CASE _eState
OF
  E_PROGRESS.PROGRESS_INIT:
    IF Execute 
    THEN
      memset(ADR(_stMsg),0,SIZEOF(_stMsg));
      _nErrorId                     := 0;
      _rValue                       := 0;
      _eState                       := E_PROGRESS.PROGRESS_BUSY;
    END_IF
END_CASE
CASE _eState
OF
  E_PROGRESS.PROGRESS_BUSY:
    IF (_AxisRef.NcToPlc.AxisId <> 0)
    THEN
      _stMsg.eType                  := E_MessageType.eMessageVerbose;
      _stMsg.eDevice                := e_Device.Axis + (_AxisRef.NcToPlc.AxisId);
      _stMsg.eSubdevice             := e_Subdevice.AxisStartUp;
      _stMsg.iErrorNumber           := 0;
      _stMsg.sText                  := concat('StartUp NcAxisId: ', TO_STRING(_AxisRef.NcToPlc.AxisId));

      IF (_MessageLevel = E_MessageType.eMessageVerbose)
      THEN
        f_MessageSet(_stMsg);
      END_IF

      _eState                       := E_PROGRESS.PROGRESS_STARTUP;
    END_IF
END_CASE
CASE _eState
OF
  E_PROGRESS.PROGRESS_STARTUP:
    _fbADSRead(
              NETID                 := '', 
              PORT                  := 501, 
              IDXGRP                := (16#5000 + _AxisRef.NcToPlc.AxisId), 
              IDXOFFS               := 16#00000003, // offset for encoder type
              LEN                   := SIZEOF(_nEncoderType), 
              DESTADDR              := ADR(_nEncoderType),
              TMOUT                 := T#200MS,
              READ                  := FALSE);

    // clear required ADS information
    _sAxisName      := _sName       := 'NO NAME';
    _sEncoderType   := _sEncoder    := 'NO TYPE';
    _nEncoderType   := _uiEncType   :=  0;

    _eState                         := E_PROGRESS.PROGRESS_PREPARE;
END_CASE
CASE _eState
OF
  E_PROGRESS.PROGRESS_PREPARE:
    _fbADSRead(
              NETID                 := '', 
              PORT                  := 501, 
              IDXGRP                := (16#5000 + _AxisRef.NcToPlc.AxisId), 
              IDXOFFS               := 16#00000003, // offset for encoder type
              LEN                   := SIZEOF(_nEncoderType), 
              DESTADDR              := ADR(_nEncoderType),
              TMOUT                 := T#200MS,
              READ                  := TRUE);

    IF (_fbADSRead.ERR)
    THEN
      _nErrorId                     := _fbAdsRead.ERRID;

      _stMsg.eType                  := E_MessageType.eMessageError;
      _stMsg.eDevice                := e_Device.Axis + (_AxisRef.NcToPlc.AxisId);
      _stMsg.eSubdevice             := e_Subdevice.AxisStartUp;
      _stMsg.iErrorNumber           := _nErrorId;
      _stMsg.sText                  := 'StartUp Ads Error Read Encoder Type';

      f_MessageSet(_stMsg);
      _eState                       := E_PROGRESS.PROGRESS_ERROR;

    ELSIF (_nEncoderType <> 0)
    THEN
      _uiEncType  := _eEncoderType  := _nEncoderType;
      _sEncoder   := _sEncoderType  := TO_STRING(_eEncoderType);

      _stMsg.eType                  := E_MessageType.eMessageInfo;
      _stMsg.eDevice                := e_Device.Axis + (_AxisRef.NcToPlc.AxisId);
      _stMsg.eSubdevice             := e_Subdevice.AxisStartUp;
      _stMsg.iErrorNumber           := 0;
      _stMsg.sText                  := concat('Encoder Type: ', _sEncoder);

      IF (_MessageLevel > E_MessageType.eMessageError)
      THEN
        f_MessageSet(_stMsg);
      END_IF

      _eState                       := E_PROGRESS.PROGRESS_CHECK;
    END_IF
END_CASE
CASE _eState
OF
  E_PROGRESS.PROGRESS_CHECK:
    _fbADSRead(
            NETID                   := '', 
            PORT                    := 501, 
            IDXGRP                  := (16#4000 + _AxisRef.NcToPlc.AxisId), 
            IDXOFFS                 := 16#00000002, // offset for axis name
            LEN                     := SIZEOF(_sAxisName), 
            DESTADDR                := ADR(_sAxisName),
            READ                    := FALSE);

    _eState                         := E_PROGRESS.PROGRESS_OCCUPIED;
END_CASE
CASE _eState
OF
  E_PROGRESS.PROGRESS_OCCUPIED:
    _fbADSRead(
            NETID                   := '', 
            PORT                    := 501, 
            IDXGRP                  := (16#4000 + _AxisRef.NcToPlc.AxisId), 
            IDXOFFS                 := 16#00000002, // offset for axis name
            LEN                     := SIZEOF(_sAxisName), 
            DESTADDR                := ADR(_sAxisName),
            READ                    := TRUE);

    IF (_fbADSRead.ERR)
    THEN
      _nErrorId                     := _fbAdsRead.ERRID;

      _stMsg.eType                  := E_MessageType.eMessageError;
      _stMsg.eDevice                := e_Device.Axis + (_AxisRef.NcToPlc.AxisId);;
      _stMsg.eSubdevice             := e_Subdevice.AxisStartUp;
      _stMsg.iErrorNumber           := _nErrorId;
      _stMsg.sText                  := 'StartUp Ads Error Read Axis Name';

      f_MessageSet(_stMsg);
      _eState                       := E_PROGRESS.PROGRESS_ERROR;

    ELSIF (_sAxisName <> 'NO NAME')
    THEN
      _sName                        := _sAxisName;

      _stMsg.eType                  := E_MessageType.eMessageInfo;
      _stMsg.eDevice                := e_Device.Axis + (_AxisRef.NcToPlc.AxisId);;
      _stMsg.eSubdevice             := e_Subdevice.AxisStartUp;
      _stMsg.iErrorNumber           := 0;
      _stMsg.sText                  := concat('Axis Name: ', _sName);

      IF (_MessageLevel > E_MessageType.eMessageError)
      THEN
        f_MessageSet(_stMsg);
      END_IF

      _eState                       := E_PROGRESS.PROGRESS_WORKING;
    END_IF
END_CASE
CASE _eState
OF
  E_PROGRESS.PROGRESS_WORKING:
    _eState                         := E_PROGRESS.PROGRESS_DONE;
END_CASE

StartUp                             := _eState;
END_METHOD

METHOD Stop : E_PROGRESS
VAR_INPUT
  Execute           : BOOL;
  Dec               : LREAL;
  Jerk              : LREAL;

END_VAR
VAR_INST
  _eState           : E_PROGRESS;
  _rValue           : LREAL;
  _stMsg            : ST_Message;
END_VAR
IF NOT (__ISVALIDREF(_AxisRef)) THEN  Stop  := E_PROGRESS.PROGRESS_ERROR; RETURN; END_IF
IF NOT Execute THEN _eState := E_PROGRESS.PROGRESS_INIT; END_IF

CASE _eState
OF
  E_PROGRESS.PROGRESS_INIT:
    IF Execute 
    THEN
      memset(ADR(_stMsg),0,SIZEOF(_stMsg));
      _nErrorId                     := 0;
      _rValue                       := 0;
      _eState                       := E_PROGRESS.PROGRESS_BUSY;
    END_IF
END_CASE
CASE _eState
OF
  E_PROGRESS.PROGRESS_BUSY:
    _eState                         := E_PROGRESS.PROGRESS_OCCUPIED;
    _fbStop(
              Axis                  := _AxisRef, 
              Execute               := FALSE, 
              Deceleration          := Dec, 
              Jerk                  := Jerk);
END_CASE
CASE _eState
OF
  E_PROGRESS.PROGRESS_OCCUPIED:
    _fbStop(
              Axis                  := _AxisRef, 
              Execute               := TRUE, 
              Deceleration          := Dec, 
              Jerk                  := Jerk);

    IF _fbStop.Error
    THEN
        _nErrorId                   := _fbStop.ErrorID;

        _stMsg.eType                := E_MessageType.eMessageError;
        _stMsg.eDevice              := e_Device.Axis + (_AxisRef.NcToPlc.AxisId);
        _stMsg.eSubdevice           := e_SubDevice.fbStop;
        _stMsg.iErrorNumber         := _nErrorId;

        f_MessageSet(_stMsg);
        _fbStop(
              Axis                  := _AxisRef, 
              Execute               := FALSE);

      _eState                       := E_PROGRESS.PROGRESS_ERROR;

    ELSE
      IF _fbStop.Done OR
         _AxisRef.Status.NotMoving
      THEN
        _eState                     := E_PROGRESS.PROGRESS_WORKING;

      ELSIF _fbStop.CommandAborted
      THEN
        _eState                     := E_PROGRESS.PROGRESS_BUSY;
      END_IF
    END_IF
END_CASE
CASE _eState
OF
  E_PROGRESS.PROGRESS_WORKING:
    _fbStop(
              Axis                  := _AxisRef, 
              Execute               := FALSE);

    _eState                         := E_PROGRESS.PROGRESS_DONE;
END_CASE


Stop                                := _eState;
END_METHOD

METHOD Template : E_PROGRESS
VAR_INPUT
  Execute           : BOOL;
END_VAR
VAR_INST
  _eState           : E_PROGRESS;
  _rValue           : LREAL;
  _udiErr           : UDINT;
  _stMsg            : ST_Message;


END_VAR
IF NOT (__ISVALIDREF(_AxisRef)) THEN _eState := E_PROGRESS.ERROR; END_IF
IF NOT Execute THEN _eState := E_PROGRESS.INIT; END_IF

CASE _eState
OF
  E_PROGRESS.INIT:
    IF Execute 
    THEN
      memset(ADR(_stMsg),0,SIZEOF(_stMsg));
      _udiErr                       := 0;
      _rValue                       := 0;
      _eState                       := E_PROGRESS.BUSY;
    END_IF
END_CASE
CASE _eState
OF
  E_PROGRESS.BUSY:
    _eState                         := E_PROGRESS.STARTUP;
END_CASE
CASE _eState
OF
  E_PROGRESS.STARTUP:
    _eState                       := E_PROGRESS.PREPARE;
END_CASE
CASE _eState
OF
  E_PROGRESS.PREPARE:
    _eState                         := E_PROGRESS.READY;
END_CASE
CASE _eState
OF
  E_PROGRESS.READY:
    _eState                         := E_PROGRESS.WAITING;
END_CASE
CASE _eState
OF
  E_PROGRESS.WAITING:
    _eState                         := E_PROGRESS.WORKING;
END_CASE
CASE _eState
OF
  E_PROGRESS.WORKING:
    _eState                         := E_PROGRESS.DONE;
END_CASE

Template_1 := _eState;
END_METHOD

METHOD WriteParameter : E_PROGRESS
VAR_INPUT
  Execute           : BOOL;
  Value             : LREAL;
  ParameterNumber   : Tc2_MC2.MC_AxisParameter;
END_VAR
VAR_INST
  _eState           : E_PROGRESS;
  _nParameter       : Tc2_MC2.MC_AxisParameter;
  _rValue           : LREAL;
  _stMsg            : ST_Message;
END_VAR
IF NOT (__ISVALIDREF(_AxisRef)) THEN  WriteParameter  := E_PROGRESS.PROGRESS_ERROR; RETURN; END_IF
IF NOT Execute THEN _eState := E_PROGRESS.PROGRESS_INIT; END_IF

CASE _eState
OF
  E_PROGRESS.PROGRESS_INIT:
    IF Execute 
    THEN
      memset(ADR(_stMsg),0,SIZEOF(_stMsg));
      _nParameter                   := 0;
      _nErrorId                     := 0;
      _rValue                       := 0;
      _eState                       := E_PROGRESS.PROGRESS_BUSY;
    END_IF
END_CASE
CASE _eState
OF
  E_PROGRESS.PROGRESS_BUSY:
    _eState                         := E_PROGRESS.PROGRESS_STARTUP;
    _nParameter                     := ParameterNumber;

    _fbWriteParameter(
                    Axis            := _AxisRef, 
                    Execute         := FALSE, 
                    ParameterNumber := ParameterNumber, 
                    Value           := Value);
END_CASE
CASE _eState
OF
  E_PROGRESS.PROGRESS_STARTUP:
    _eState                         := E_PROGRESS.PROGRESS_OCCUPIED;
    _fbWriteParameter(
                    Axis            := _AxisRef, 
                    Execute         := TRUE, 
                    ParameterNumber := ParameterNumber, 
                    Value           := Value);

END_CASE
CASE _eState
OF
  E_PROGRESS.PROGRESS_OCCUPIED:
    _fbWriteParameter(
                    Axis            := _AxisRef, 
                    ParameterNumber := ParameterNumber, 
                    Value           := Value);

    IF _fbWriteParameter.Error
    THEN
      _nErrorId                     := _fbWriteParameter.ErrorID;

      _stMsg.eType                  := E_MessageType.eMessageError;
      _stMsg.eDevice                := e_Device.Axis + (_AxisRef.NcToPlc.AxisId);
      _stMsg.eSubdevice             := e_SubDevice.fbWriteParameter;
      _stMsg.iErrorNumber           := _nErrorId;

      f_MessageSet(_stMsg);

      _fbWriteParameter(
                    Axis            := _AxisRef,
                    Execute         := FALSE, 
                    ParameterNumber := ParameterNumber, 
                    Value           := Value);


      _eState                       := E_PROGRESS.PROGRESS_ERROR;
    ELSE
      IF _fbWriteParameter.Done
      THEN
        _rValue                     := _fbWriteParameter.Value;
        _eState                     := E_PROGRESS.PROGRESS_WORKING;
      END_IF
    END_IF

END_CASE
CASE _eState
OF
  E_PROGRESS.PROGRESS_WORKING:
    _fbWriteParameter(
                    Axis            := _AxisRef,
                    Execute         := FALSE, 
                    ParameterNumber := ParameterNumber, 
                    Value           := Value);
    _eState                         := E_PROGRESS.PROGRESS_DONE;
END_CASE


WriteParameter                      := _eState;
END_METHOD

METHOD WriteParameterPersistent : E_PROGRESS
VAR_INPUT
  Execute           : BOOL;
  Value             : LREAL;
  ParameterNumber   : Tc2_MC2.MC_AxisParameter;
END_VAR
VAR_INST
  _eState           : E_PROGRESS;
  _rValue           : LREAL;
  _stMsg            : ST_Message;
END_VAR
IF NOT (__ISVALIDREF(_AxisRef)) THEN  WriteParameterPersistent  := E_PROGRESS.PROGRESS_ERROR; RETURN; END_IF
IF NOT Execute THEN _eState := E_PROGRESS.PROGRESS_INIT; END_IF

CASE _eState
OF
  E_PROGRESS.PROGRESS_INIT:
    IF Execute 
    THEN
      memset(ADR(_stMsg),0,SIZEOF(_stMsg));
      _nErrorId                     := 0;
      _rValue                       := 0;
      _eState                       := E_PROGRESS.PROGRESS_BUSY;
    END_IF
END_CASE
CASE _eState
OF
  E_PROGRESS.PROGRESS_BUSY:
    _eState                         := E_PROGRESS.PROGRESS_STARTUP;
    _fbWriteParameterPersist(
                    Axis            := _AxisRef, 
                    Execute         := FALSE, 
                    ParameterNumber := ParameterNumber, 
                    Value           := Value);
END_CASE
CASE _eState
OF
  E_PROGRESS.PROGRESS_STARTUP:
    _eState                         := E_PROGRESS.PROGRESS_OCCUPIED;
    _fbWriteParameterPersist(
                    Axis            := _AxisRef, 
                    Execute         := TRUE, 
                    ParameterNumber := ParameterNumber, 
                    Value           := Value);

END_CASE
CASE _eState
OF
  E_PROGRESS.PROGRESS_OCCUPIED:
    _fbWriteParameterPersist(
                    Axis            := _AxisRef, 
                    ParameterNumber := ParameterNumber, 
                    Value           := Value);

    IF (_fbWriteParameterPersist.Error)
    THEN
      _nErrorId                     := _fbWriteParameterPersist.ErrorID;

      _stMsg.eType                  := E_MessageType.eMessageError;
      _stMsg.eDevice                := e_Device.Axis + (_AxisRef.NcToPlc.AxisId);
      _stMsg.eSubdevice             := e_SubDevice.fbWriteParameterPersistent;
      _stMsg.iErrorNumber           := _nErrorId;

      f_MessageSet(_stMsg);

      _fbWriteParameterPersist(
                    Axis            := _AxisRef,
                    Execute         := FALSE, 
                    ParameterNumber := ParameterNumber, 
                    Value           := Value);


      _eState                       := E_PROGRESS.PROGRESS_ERROR;
    ELSE
      IF (_fbWriteParameterPersist.Done)
      THEN
        _rValue                     := _fbWriteParameterPersist.Value;
        _eState                     := E_PROGRESS.PROGRESS_WORKING;
      END_IF
    END_IF

END_CASE
CASE _eState
OF
  E_PROGRESS.PROGRESS_WORKING:
    _fbWriteParameterPersist(
                    Axis            := _AxisRef,
                    Execute         := FALSE, 
                    ParameterNumber := ParameterNumber, 
                    Value           := Value);

    _eState                         := E_PROGRESS.PROGRESS_DONE;
END_CASE


WriteParameterPersistent            := _eState;
END_METHOD

END_FUNCTION_BLOCK

// ---- FUNCTIONS/TRIGGER_BOX/FB_TriggerBox.TcPOU
//-----------------------------------------------------------------------------------------------------------
// TriggerBox
//
// HAUD
// 17.07.2024
// - init: ALL outputs will be switched of 
// - controlled via ST_TriggerBox
// - position and timestamp based setting of digital output
// - feedback from digital input with timestamp
// - AxisPosition at timestamp as result
//-----------------------------------------------------------------------------------------------------------
FUNCTION_BLOCK FB_TriggerBox EXTENDS FB_Xfc
VAR
  _Ctrl             : REFERENCE TO ARRAY[1..MAX_TRIGGER_BOX] OF ST_CTRL_TRIGGER;
  _State            : REFERENCE TO ARRAY[1..MAX_TRIGGER_BOX] OF ST_STATE_TRIGGER;

  _Input            : POINTER TO ARRAY[1..MAX_TRIGGER_BOX]   OF ST_DC_Input;
  _Output_2252      : POINTER TO ARRAY[1..MAX_TRIGGER_BOX]   OF ST_DC_Output;

  _Index            : UDINT;
  _AxisId           : UDINT;
  _AxisIndex        : UDINT;

  _CtrlLocal        : ST_CTRL_TRIGGER;
  _McDirection      : Tc2_MC2.MC_Direction;

  _eStateProgress   : E_PROGRESS;
  _eResult          : E_PROGRESS;
  _eInit            : E_PROGRESS;

  _rtrigEnable      : Tc2_Standard.R_TRIG;
  _rtrigInit        : Tc2_Standard.R_TRIG;
  _TrigCount        : UDINT := 1; // counter for active index in _stCtrl.TriggerPosition[]

  _CurrentTime      : ULINT;      // current DC time 64 bit
  _CurrentTimeShort : UDINT;      // current DC time 32 bit
  _LatchTime        : UDINT;
  _SwitchTime       : ULINT;      // DC time for output at _stCtrl.TriggerPosition[_TrigCount]
  _SafeCycles       : BYTE := 3;  // cycles needed to get the SwitchTime onto the terminal/output

  _bError           : BOOL;
  _stMsg            : ST_Message;
  _MessageLevel     : E_MessageType;
END_VAR

PROPERTY Ctrl : REFERENCE TO ARRAY [1..MAX_TRIGGER_BOX] OF ST_CTRL_TRIGGER
SET
_Ctrl REF= Ctrl;
END_SET
END_PROPERTY

METHOD Cycle : BOOL
VAR_INPUT
END_VAR
//-----------------------------------------------------------------------------
// trigger detection
//-----------------------------------------------------------------------------
_rtrigEnable(CLK                := _Ctrl[_Index].Control.Enable);
_rtrigInit(  CLK                := _Ctrl[_Index].Control.Init);
//-----------------------------------------------------------------------------
// forced init
//-----------------------------------------------------------------------------
IF _rtrigInit.Q THEN _eInit     := E_PROGRESS.PROGRESS_INVALID; END_IF
//-----------------------------------------------------------------------------
// clear state
//-----------------------------------------------------------------------------
IF NOT _Ctrl[_Index].Control.Enable 
THEN 
  _eStateProgress               := E_PROGRESS.PROGRESS_INVALID;

  _State[_Index].State          := TO_UINT(_eStateProgress);
END_IF

_eDeviceFunction                := e_Device.XfcTriggerBox + _Index;

_CurrentTime                    := Tc2_EtherCAT.F_GetCurDcTickTime64();
_CurrentTimeShort               := TO_UDINT(_CurrentTime AND 16#FFFFFFFF);

_State[_Index].Init             := TO_UINT(_eInit);

IF NOT (_eInit = E_PROGRESS.PROGRESS_DONE)
THEN
  _eInit                        := Init();
  RETURN;
END_IF
//-----------------------------------------------------------------------------
// TriggerBox execution
//-----------------------------------------------------------------------------
CASE _eStateProgress
OF
  E_PROGRESS.PROGRESS_INVALID:  // check input data
    IF _rtrigEnable.Q
    THEN
      _State[_Index].State      := TO_UINT(E_PROGRESS.PROGRESS_BUSY);

      _bError                   := FALSE;
      _TrigCount                := 1;     // initialize trigger counter for output on TriggerPositions
      _eStateProgress           := E_PROGRESS.PROGRESS_INIT;

      _CtrlLocal                := _Ctrl[_Index];
      _AxisId                   := _CtrlLocal.AxisId;
      _AxisIndex                := GetIndex(_AxisId);

      _eResult                  := TimeToPosition(FALSE, _AxisId, 0.0, _MessageLevel);
      _eResult                  := WaitForPosition(FALSE, _AxisId, _CtrlLocal.TriggerPosition[_TrigCount], _MessageLevel);

      IF NOT (_AxisIndex > 0) OR NOT (_AxisId > 0)
      THEN
        _bError                 := TRUE;
        _stMsg.iErrorNumber     := 10;
        _stMsg.eSubdevice       := XfcTriggerStart;
        _stMsg.sText            := 'AxisId Invalid ';
        _eStateProgress         := E_PROGRESS.PROGRESS_STILL_WORKING;
      END_IF

      IF NOT (_CtrlLocal.TriggerCount > 0) OR
         NOT (_CtrlLocal.TriggerCount < TO_UDINT(MAX_TRIGGER_COUNT+1))
      THEN
        _bError                 := TRUE;
        _stMsg.iErrorNumber     := 11;
        _stMsg.eSubdevice       := XfcTriggerStart;
        _stMsg.sText            := 'TriggerCount Invalid ';
        _eStateProgress         := E_PROGRESS.PROGRESS_STILL_WORKING;
      END_IF

      IF (_MessageLevel = E_MessageType.eMessageVerbose)
      THEN
        _stMsg.eType            := E_MessageType.eMessageVerbose;
        _stMsg.eDevice          := _eDeviceFunction;
        _stMsg.eSubdevice       := e_Subdevice.XfcTriggerStart;
        _stMsg.iErrorNumber     := _CurrentTime;
        _stMsg.sText            := concat(TO_STRING(_eStateProgress), ': ');
        _stMsg.sText            := concat(_stMsg.sText, TO_STRING(e_Device.XfcAxis));
        _stMsg.sText            := concat(_stMsg.sText, '_ID_');
        _stMsg.sText            := concat(_stMsg.sText, TO_STRING(_AxisId));

        f_MessageSet(_stMsg);
      END_IF
    END_IF


  E_PROGRESS.PROGRESS_INIT:
    _eDeviceAxis                := e_Device.XfcAxis + (_CtrlLocal.AxisId);
    _eResult                    := WaitForPosition(TRUE, _AxisId, _CtrlLocal.TriggerPosition[_TrigCount], _MessageLevel);

    IF (_eResult = E_PROGRESS.PROGRESS_ERROR)
    THEN
      _bError                   := TRUE;
      _stMsg.iErrorNumber       := 16;
      _stMsg.eSubdevice         := XfcWaitForPosition;
      _stMsg.sText              := 'Position not reachable ';
      _eStateProgress           := E_PROGRESS.PROGRESS_STILL_WORKING;

    ELSIF (_eResult = E_PROGRESS.PROGRESS_DONE)
    THEN
      _eStateProgress           := E_PROGRESS.PROGRESS_BUSY;

      IF (_MessageLevel = E_MessageType.eMessageVerbose)
      THEN
        _stMsg.eType            := E_MessageType.eMessageVerbose;
        _stMsg.eDevice          := _eDeviceFunction;
        _stMsg.eSubdevice       := e_Subdevice.XfcWaitForPosition;
        _stMsg.iErrorNumber     := _CurrentTime;
        _stMsg.sText            := concat(TO_STRING(_eStateProgress), ': ');
        _stMsg.sText            := concat(_stMsg.sText, TO_STRING(_XfcDurationToPosition[_AxisIndex]));

        f_MessageSet(_stMsg);
      END_IF
    END_IF
END_CASE
//-----------------------------------------------------------------------------
//-----------------------------------------------------------------------------
CASE _eStateProgress
OF
  E_PROGRESS.PROGRESS_BUSY:
    _eResult                    := TimeToPosition(TRUE, _AxisId, _CtrlLocal.TriggerPosition[_TrigCount], _MessageLevel);

    IF (_eResult = E_PROGRESS.PROGRESS_ERROR)
    THEN
      TimeToPosition(FALSE, _AxisId, _CtrlLocal.TriggerPosition[_TrigCount], _MessageLevel);

      _bError                   := TRUE;
      _stMsg.iErrorNumber       := 15;
      _stMsg.sText              := concat('Get TimeToPosition ', TO_STRING(_CtrlLocal.TriggerPosition[_TrigCount]));
      _stMsg.sText              := concat(_stMsg.sText, ' ');
      _eStateProgress           := E_PROGRESS.PROGRESS_STILL_WORKING;

    ELSIF (_eResult = E_PROGRESS.PROGRESS_DONE)
    THEN
      TimeToPosition(FALSE, _AxisId, _CtrlLocal.TriggerPosition[_TrigCount], _MessageLevel);

      _SwitchTime               := _CurrentTime + TO_ULINT(_XfcDurationToPosition[_AxisIndex]);
      _eResult                  := SwitchOn_2252(FALSE, _SwitchTime, 3);
 
      IF (_MessageLevel = E_MessageType.eMessageVerbose)
      THEN
        _stMsg.eType            := E_MessageType.eMessageVerbose;
        _stMsg.eDevice          := _eDeviceFunction;
        _stMsg.eSubdevice       := e_Subdevice.XfcTimeToPosition;
        _stMsg.iErrorNumber     := _SwitchTime;
        _stMsg.sText            := concat(TO_STRING(_eStateProgress), ': ');
        _stMsg.sText            := concat(_stMsg.sText, TO_STRING(_XfcDurationToPosition[_AxisIndex]));

        f_MessageSet(_stMsg);
      END_IF
      _eStateProgress           := E_PROGRESS.PROGRESS_PREPARE;
    END_IF
END_CASE
//-----------------------------------------------------------------------------
//-----------------------------------------------------------------------------
CASE _eStateProgress
OF
  E_PROGRESS.PROGRESS_PREPARE:
    //_State[_Index].State        := TO_UINT(_eState);
    _eResult                    := SwitchOn_2252(TRUE, _SwitchTime, 3);


    IF (_CtrlLocal.Control.NoFeedback)
    THEN
      IF (_eResult = E_PROGRESS.PROGRESS_ERROR)
      THEN
        _bError                 := TRUE;
        _stMsg.iErrorNumber     := 12;
        _stMsg.eSubdevice       := XfcSwitchOn_2252;
        _stMsg.sText            := 'NO_FEEDBACK: Switch Time in the past ';
        _eStateProgress         := E_PROGRESS.PROGRESS_STILL_WORKING;

      ELSIF (_eResult = E_PROGRESS.PROGRESS_DONE)
      THEN
        _eStateProgress         := E_PROGRESS.PROGRESS_CHECK;
      END_IF

    ELSIF (_eResult = E_PROGRESS.PROGRESS_ERROR)
    THEN
        _bError                 := TRUE;
        _stMsg.iErrorNumber     := 13;
        _stMsg.eSubdevice       := XfcSwitchOn_2252;
        _stMsg.sText            := 'Switch Time in the past ';
        _eStateProgress         := E_PROGRESS.PROGRESS_STILL_WORKING;
    END_IF

    IF (_Input^[_Index].Input) OR
       (_Input^[_Index].LatchPositive >= _SwitchTime)
    THEN
      _LatchTime                := TO_UDINT(_Input^[_Index].LatchPositive AND 16#FFFFFFFF);

      IF (_MessageLevel = E_MessageType.eMessageVerbose)
      THEN
        _stMsg.eType            := E_MessageType.eMessageVerbose;
        _stMsg.eDevice          := _eDeviceFunction;
        _stMsg.eSubdevice       := e_Subdevice.XfcLatchPosition;
        _stMsg.iErrorNumber     := _LatchTime;
        _stMsg.sText            := concat(TO_STRING(_eStateProgress), ': ');
        _stMsg.sText            := concat(_stMsg.sText, TO_STRING(_eDeviceAxis));

        f_MessageSet(_stMsg);
      END_IF
      _eStateProgress           := E_PROGRESS.PROGRESS_STARTUP;
      _eResult                  := PositionAtTime(FALSE, _CtrlLocal.AxisId, 0, _MessageLevel);
      _eResult                  := SwitchOn_2252(FALSE, _SwitchTime, 3);
    END_IF
END_CASE
//-----------------------------------------------------------------------------
//-----------------------------------------------------------------------------
CASE _eStateProgress
OF
  E_PROGRESS.PROGRESS_STARTUP:
    //_State[_Index].State        := TO_UINT(_eState);
    _eResult                    := PositionAtTime(TRUE, _CtrlLocal.AxisId, _LatchTime, _MessageLevel);

    IF (_eResult = E_PROGRESS.PROGRESS_ERROR)
    THEN
      _bError                   := TRUE;
      _stMsg.iErrorNumber       := 14;
      _stMsg.sText              := 'PositionAtTime LatchPositive ';
      _eStateProgress           := E_PROGRESS.PROGRESS_STILL_WORKING;
      _eResult                  := PositionAtTime(FALSE, _CtrlLocal.AxisId, 0, _MessageLevel);

    ELSIF (_eResult = E_PROGRESS.PROGRESS_DONE)
    THEN
      _State[_Index].FlashPosition[_TrigCount]  := _XfcRecordedPosition[_AxisIndex];

      IF (_MessageLevel = E_MessageType.eMessageVerbose)
      THEN
        _stMsg.eType            := E_MessageType.eMessageVerbose;
        _stMsg.eDevice          := _eDeviceFunction;
        _stMsg.eSubdevice       := e_Subdevice.XfcRecordedPosition;
        _stMsg.iErrorNumber     := _LatchTime;
        _stMsg.sText            := concat(TO_STRING(_eStateProgress), ': ');
        _stMsg.sText            := concat(_stMsg.sText, TO_STRING(_XfcRecordedPosition[_AxisIndex]));

        f_MessageSet(_stMsg);
      END_IF
      _eStateProgress           := E_PROGRESS.PROGRESS_CHECK;
      _eResult                  := PositionAtTime(FALSE, _CtrlLocal.AxisId, 0, _MessageLevel);
      _eResult                  := SwitchOff_2252(FALSE, 3);
    END_IF
END_CASE
//-----------------------------------------------------------------------------
//-----------------------------------------------------------------------------
CASE _eStateProgress
OF
  E_PROGRESS.PROGRESS_CHECK:
    _State[_Index].State        := TO_UINT(_eStateProgress) + TO_UINT(_TrigCount);
    _eResult                    := SwitchOff_2252(TRUE, 4);
    IF (_eResult = E_PROGRESS.PROGRESS_DONE)
    THEN
      _eResult                  := SwitchOff_2252(FALSE, 4);
      _TrigCount                := _TrigCount + 1;

      IF (_TrigCount > _CtrlLocal.TriggerCount)
      THEN
        _eStateProgress         := E_PROGRESS.PROGRESS_OCCUPIED;
      ELSE
        _eStateProgress         := E_PROGRESS.PROGRESS_INIT;
        _eResult                := WaitForPosition(FALSE, _AxisId, _CtrlLocal.TriggerPosition[_TrigCount], _MessageLevel);
      END_IF
    END_IF
END_CASE
//-----------------------------------------------------------------------------
//-----------------------------------------------------------------------------
CASE _eStateProgress
OF
  E_PROGRESS.PROGRESS_OCCUPIED:
    _eStateProgress             := E_PROGRESS.PROGRESS_WORKING;
END_CASE
//-----------------------------------------------------------------------------
//-----------------------------------------------------------------------------
CASE _eStateProgress
OF
  E_PROGRESS.PROGRESS_WORKING:
    _eStateProgress             := E_PROGRESS.PROGRESS_STILL_WORKING;
END_CASE
//-----------------------------------------------------------------------------
//-----------------------------------------------------------------------------
CASE _eStateProgress
OF
  E_PROGRESS.PROGRESS_STILL_WORKING:
    IF NOT _bError
    THEN
      _eStateProgress           := E_PROGRESS.PROGRESS_DONE;

      IF (_MessageLevel > E_MessageType.eMessageWarning)
      THEN
        _stMsg.eType            := E_MessageType.eMessageInfo;
        _stMsg.eDevice          := _eDeviceFunction;
        _stMsg.eSubdevice       := e_Subdevice.XfcTriggerOut;
        _stMsg.iErrorNumber     := _CurrentTime;
        _stMsg.sText            := concat(TO_STRING(_eStateProgress), ': ');
        _stMsg.sText            := concat(_stMsg.sText, TO_STRING(e_Device.XfcAxis));
        _stMsg.sText            := concat(_stMsg.sText, '_ID_');
        _stMsg.sText            := concat(_stMsg.sText, TO_STRING(_AxisId));
        f_MessageSet(_stMsg);
      END_IF
      _State[_Index].State      := TO_UINT(_eStateProgress);
    ELSE
      _eStateProgress           := E_PROGRESS.PROGRESS_ERROR;

      _stMsg.eType              := E_MessageType.eMessageError;
      _stMsg.eDevice            := _eDeviceFunction;
      _stMsg.eSubdevice         := e_Subdevice.XfcTriggerOut;
      _stMsg.sText              := concat(_stMsg.sText, TO_STRING(_eStateProgress));

      f_MessageSet(_stMsg);

      _State[_Index].State      := TO_UINT(_eStateProgress) + TO_UINT(_stMsg.iErrorNumber);
    END_IF
END_CASE
END_METHOD

PROPERTY Index : udint
GET
Index := _Index;
END_GET
SET
_Index := Index;
END_SET
END_PROPERTY

METHOD Init : E_PROGRESS
VAR_INST
  _eState         : E_PROGRESS;
  _eResult        : E_PROGRESS;

  _stMsg          : ST_Message;
  _bError         : BOOL;
  _udiErrorId     : UDINT;

  _nIdx           : udint;
END_VAR

_stMsg.eDevice                  := _eDeviceFunction;
_stMsg.eSubdevice               := XfcInit;


CASE _eInit
OF
  E_PROGRESS.PROGRESS_INVALID:
    _eState                     := E_PROGRESS.PROGRESS_INIT;
    _bError                     := FALSE;
    _udiErrorId                 := 0;
END_CASE
//-----------------------------------------------------------------------------
//-----------------------------------------------------------------------------
CASE _eState
OF
  E_PROGRESS.PROGRESS_INIT:
    _eResult                    := SwitchOff_2252(FALSE, 2);
    _eState                     := E_PROGRESS.PROGRESS_BUSY;

      IF (_MessageLevel = E_MessageType.eMessageVerbose)
      THEN
        _stMsg.eType            := E_MessageType.eMessageVerbose;
        _stMsg.iErrorNumber     := 0;
        _stMsg.sText            := TO_STRING(_eState);

        f_MessageSet(_stMsg);
      END_IF

  //-----------------------------------------------------------------------------
  // clear output terminals 2252
  //-----------------------------------------------------------------------------
  E_PROGRESS.PROGRESS_BUSY:
    _eResult                    := SwitchOff_2252(TRUE, 10);

    IF (_eResult = E_PROGRESS.PROGRESS_DONE)
    THEN
      IF (_Index > 0) AND
         (_Index < MAX_TRIGGER_BOX+1)
      THEN
        FOR _nIdx := 1 TO MAX_TRIGGER_COUNT
        DO
          _State[_Index].FlashPosition[_nIdx] := 0.0;
        END_FOR
      END_IF

      _eState                   := E_PROGRESS.PROGRESS_PREPARE;
      _eResult                  := SwitchOff_2252(FALSE, 10);
    END_IF
END_CASE
//-----------------------------------------------------------------------------
// reserve states for future timestamp outputs with dedicated switch off
//-----------------------------------------------------------------------------
CASE _eState
OF
  E_PROGRESS.PROGRESS_PREPARE:
    _eState                     := E_PROGRESS.PROGRESS_STARTUP;
END_CASE
//-----------------------------------------------------------------------------
//-----------------------------------------------------------------------------
CASE _eState
OF
  E_PROGRESS.PROGRESS_STARTUP:
    _eState                     := E_PROGRESS.PROGRESS_CHECK;
END_CASE
//-----------------------------------------------------------------------------
//-----------------------------------------------------------------------------
CASE _eState
OF
  E_PROGRESS.PROGRESS_CHECK:
    _eState                     := E_PROGRESS.PROGRESS_OCCUPIED;
END_CASE
//-----------------------------------------------------------------------------
//-----------------------------------------------------------------------------
CASE _eState
OF
  E_PROGRESS.PROGRESS_OCCUPIED:
    _eState                     := E_PROGRESS.PROGRESS_WORKING;
END_CASE
//-----------------------------------------------------------------------------
//-----------------------------------------------------------------------------
CASE _eState
OF
  E_PROGRESS.PROGRESS_WORKING:
    _eState                     := E_PROGRESS.PROGRESS_STILL_WORKING;
END_CASE
//-----------------------------------------------------------------------------
//-----------------------------------------------------------------------------
CASE _eState
OF
  E_PROGRESS.PROGRESS_STILL_WORKING:
    IF NOT _bError
    THEN
      _eState                   := E_PROGRESS.PROGRESS_DONE;

      IF (_MessageLevel > E_MessageType.eMessageWarning)
      THEN
        _stMsg.eType            := E_MessageType.eMessageInfo;
        _stMsg.iErrorNumber     := 0;
        _stMsg.sText            := TO_STRING(_eState);
      END_IF
    ELSE
      _eState                   := E_PROGRESS.PROGRESS_ERROR;

      _stMsg.eType              := E_MessageType.eMessageError;
      _stMsg.iErrorNumber       := _udiErrorId;
      _stMsg.sText              := TO_STRING(_eState);
    END_IF
END_CASE

Init                            := _eState;
END_METHOD

PROPERTY Input : pointer TO ARRAY [1..MAX_TRIGGER_BOX] OF ST_DC_Input
SET
_Input := Input;
END_SET
END_PROPERTY

PROPERTY MessageLevel : e_messagetype
GET
MessageLevel := _MessageLevel;
END_GET
SET
_MessageLevel := MessageLevel;
END_SET
END_PROPERTY

PROPERTY Output_2252 : pointer TO ARRAY [1..MAX_TRIGGER_BOX] OF ST_DC_Output
SET
_Output_2252 := Output_2252;
END_SET
END_PROPERTY

PROPERTY State : REFERENCE TO ARRAY[1..MAX_TRIGGER_BOX] OF ST_STATE_TRIGGER
SET
_State REF= State;
END_SET
END_PROPERTY

METHOD SwitchOff_2252 : E_PROGRESS
VAR_INPUT
  Execute         : BOOL;
  DurationCycles  : UINT := 3;   // PLC cycles are counted after the output time was reached before the method returns done
END_VAR
VAR_INST
  _bError             : BOOL;
  _eState             : E_PROGRESS;

  _stMsg              : ST_Message;
  _CurrentStartTime   : ULINT;
  _nCount             : UINT;
END_VAR
IF NOT Execute THEN _eState     := E_PROGRESS.PROGRESS_INIT;  END_IF


CASE _eState
OF
  E_PROGRESS.PROGRESS_INIT:
    IF Execute
    THEN
      _nCount                   := 0;
      _bError                   := FALSE;
      _eState                   := E_PROGRESS.PROGRESS_BUSY;
      _CurrentStartTime         := Tc2_EtherCAT.F_GetCurDcTickTime64();

      _Output_2252^[_Index].nActivate     := 0;

      IF (_MessageLevel = E_MessageType.eMessageVerbose)
      THEN
        _stMsg.eType            := E_MessageType.eMessageVerbose;
        _stMsg.eDevice          := _eDeviceFunction;
        _stMsg.eSubdevice       := XfcSwitchOff_2252;
        _stMsg.iErrorNumber     := _CurrentStartTime;
        _stMsg.sText            := TO_STRING(_eState);
        f_MessageSet(_stMsg);
      END_IF
    END_IF

  E_PROGRESS.PROGRESS_BUSY:
    _Output_2252^[_Index].Ch1_Output    := FALSE;
    _Output_2252^[_Index].Ch2_Output    := FALSE;

    _Output_2252^[_Index].Ch1_Tristate  := FALSE;
    _Output_2252^[_Index].Ch2_Tristate  := FALSE;

    _Output_2252^[_Index].dcStartTime   := (_CurrentStartTime + DurationCycles*2_000_000);
    _Output_2252^[_Index].nActivate     := 0;
    _eState                             := E_PROGRESS.PROGRESS_PREPARE;


  E_PROGRESS.PROGRESS_PREPARE:
    _Output_2252^[_Index].nActivate     := 3;
    _eState                             := E_PROGRESS.PROGRESS_STARTUP;

  E_PROGRESS.PROGRESS_STARTUP:
    IF (_CurrentTime > _Output_2252^[_Index].dcStartTime)
    THEN
      //_Output_2252^[_Index].nActivate   := 0;
      _eState                           := E_PROGRESS.PROGRESS_CHECK;
    END_IF

  E_PROGRESS.PROGRESS_CHECK:
    _nCount                             := _nCount + 1;
    IF (_nCount > DurationCycles-1)
    THEN
      _Output_2252^[_Index].nActivate   := 0;
      _eState                           := E_PROGRESS.PROGRESS_STILL_WORKING;
    END_IF
END_CASE
//-----------------------------------------------------------------------------
//-----------------------------------------------------------------------------
CASE _eState
OF
  E_PROGRESS.PROGRESS_STILL_WORKING:
    IF NOT _bError
    THEN
      _eState                   := E_PROGRESS.PROGRESS_DONE;

      IF (_MessageLevel > E_MessageType.eMessageWarning)
      THEN
        _stMsg.eType            := E_MessageType.eMessageInfo;
        _stMsg.eDevice          := _eDeviceFunction;
        _stMsg.eSubdevice       := XfcSwitchOff_2252;
        _stMsg.iErrorNumber     := _CurrentTime;
        _stMsg.sText            := TO_STRING(_eState);
        f_MessageSet(_stMsg);
      END_IF
    ELSE
      _eState                   := E_PROGRESS.PROGRESS_ERROR;

      _stMsg.eType              := E_MessageType.eMessageError;
      _stMsg.eDevice            := _eDeviceFunction;
      _stMsg.eSubdevice         := XfcSwitchOff_2252;
      _stMsg.sText              := concat(_stMsg.sText, TO_STRING(_eState));

      f_MessageSet(_stMsg);
 
    END_IF
END_CASE


SwitchOff_2252                  := _eState;
END_METHOD

METHOD SwitchOn_2252 : E_PROGRESS // uses _Output[] datafield directly
VAR_INPUT
  Execute         : BOOL;
  StartTime       : ULINT;
  DurationCycles  : UINT := 3;   // PLC cycles are counted after the output time was reached before the method returns done
END_VAR
VAR_INST
  _bError             : BOOL;
  _eState             : E_PROGRESS;

  _stMsg              : ST_Message;
  _CurrentStartTime   : ULINT;
  _nCount             : UINT;
END_VAR
IF NOT Execute THEN _eState     := E_PROGRESS.PROGRESS_INIT;  END_IF


CASE _eState
OF
  E_PROGRESS.PROGRESS_INIT:
    IF Execute
    THEN
      _nCount                   := 0;
      _bError                   := FALSE;
      _eState                   := E_PROGRESS.PROGRESS_BUSY;
      _CurrentStartTime         := Tc2_EtherCAT.F_GetCurDcTickTime64();

      IF (_MessageLevel = E_MessageType.eMessageVerbose)
      THEN
        _stMsg.eType            := E_MessageType.eMessageVerbose;
        _stMsg.eDevice          := _eDeviceFunction;
        _stMsg.eSubdevice       := XfcSwitchOn_2252;
        _stMsg.iErrorNumber     := _CurrentStartTime;
        _stMsg.sText            := TO_STRING(_eState);
        f_MessageSet(_stMsg);
      END_IF

      IF NOT ((_CurrentStartTime + _SafeCycles*1_000_000) < StartTime)
      THEN
        _bError                 := TRUE;
        _stMsg.sText            := 'StartTime too close to CurrentTime ';
        _eState                 := E_PROGRESS.PROGRESS_STILL_WORKING;
      END_IF

    END_IF
END_CASE
//-----------------------------------------------------------------------------
//-----------------------------------------------------------------------------
CASE _eState
OF
  E_PROGRESS.PROGRESS_BUSY:
    _Output_2252^[_Index].Ch1_Output    := TRUE;
    _Output_2252^[_Index].Ch2_Output    := TRUE;

    _Output_2252^[_Index].Ch1_Tristate  := FALSE;
    _Output_2252^[_Index].Ch2_Tristate  := FALSE;

    _Output_2252^[_Index].dcStartTime   := StartTime;
    _Output_2252^[_Index].nActivate     := 0;
    _eState                             := E_PROGRESS.PROGRESS_PREPARE;


  E_PROGRESS.PROGRESS_PREPARE:
    _Output_2252^[_Index].nActivate     := 3;
    _eState                             := E_PROGRESS.PROGRESS_CHECK;
END_CASE
//-----------------------------------------------------------------------------
//-----------------------------------------------------------------------------
CASE _eState
OF
  E_PROGRESS.PROGRESS_STARTUP:
    IF (_CurrentTime > StartTime)
    THEN
      _Output_2252^[_Index].nActivate   := 0;
      _eState                           := E_PROGRESS.PROGRESS_CHECK;
    END_IF
END_CASE
//-----------------------------------------------------------------------------
//-----------------------------------------------------------------------------
CASE _eState
OF
  E_PROGRESS.PROGRESS_CHECK:
    _nCount                             := _nCount + 1;
    IF (_nCount > DurationCycles-1)
    THEN
      _eState                           := E_PROGRESS.PROGRESS_STILL_WORKING;
    END_IF
END_CASE
//-----------------------------------------------------------------------------
//-----------------------------------------------------------------------------
CASE _eState
OF
  E_PROGRESS.PROGRESS_STILL_WORKING:
    IF NOT _bError
    THEN
      _eState                   := E_PROGRESS.PROGRESS_DONE;

      IF (_MessageLevel > E_MessageType.eMessageWarning)
      THEN
        _stMsg.eType            := E_MessageType.eMessageInfo;
        _stMsg.eDevice          := _eDeviceFunction;
        _stMsg.eSubdevice       := XfcSwitchOn_2252;
        _stMsg.iErrorNumber     := _CurrentTime;
        _stMsg.sText            := TO_STRING(_eState);
        f_MessageSet(_stMsg);
      END_IF
    ELSE
      _eState                   := E_PROGRESS.PROGRESS_ERROR;

      _stMsg.eType              := E_MessageType.eMessageError;
      _stMsg.eDevice            := _eDeviceFunction;
      _stMsg.eSubdevice         := XfcSwitchOn_2252;
      _stMsg.sText              := concat(_stMsg.sText, TO_STRING(_eState));

      f_MessageSet(_stMsg);
 
    END_IF
END_CASE


SwitchOn_2252                   := _eState;
END_METHOD

END_FUNCTION_BLOCK

// ---- XFC/FB_Xfc.TcPOU
//-----------------------------------------------------------------------------------------------------------
// XFC base class
//
// HAUD
// 18.07.2024
// - encapsulation of XFC library: Tc2_MC2_XFC
//-----------------------------------------------------------------------------------------------------------
FUNCTION_BLOCK FB_Xfc
VAR
  _eDeviceFunction            : e_Device;
  _eDeviceAxis                : e_Device;

  _XfcTaskTime_DC             : T_DCTIME;

  _ItfAxis                    : ARRAY[1..MAX_AXIS] OF I_McAxis;

  // base function blocks per axis
  _XfcPositionAtTime          : ARRAY[1..MAX_AXIS] OF Tc2_MC2_XFC.XFC_PositionAtTime;
  _XfcTimeOfPosition          : ARRAY[1..MAX_AXIS] OF Tc2_MC2_XFC.XFC_TimeOfPosition;
  _XfcTimeToPosition          : ARRAY[1..MAX_AXIS] OF Tc2_MC2_XFC.XFC_TimeToPosition;
  _XfcTimeToModuloPosition    : ARRAY[1..MAX_AXIS] OF Tc2_MC2_XFC.XFC_TimeToModuloPosition;

  _XfcNcTimeConversionOptions : ARRAY[1..MAX_AXIS] OF ST_NcTimeConversionOptions; 
  _XfcRecordedPosition        : ARRAY[1..MAX_AXIS] OF LREAL;
  _XfcRecordedTime            : ARRAY[1..MAX_AXIS] OF T_DCTIME32;

  _XfcDurationToPosition      : ARRAY[1..MAX_AXIS] OF DINT;
  _XfcDcTimeOfPosition        : ARRAY[1..MAX_AXIS] OF T_DCTIME32;

  // inputs
  _XfcTouchProbe              : Tc2_MC2_XFC.XFC_TouchProbe;
  _XfcTouchProbeEL1258        : Tc2_MC2_XFC.XFC_EL1258_TouchProbe;

  // input datatypes
  _XfcTouchProbeOptions       : Tc2_MC2_XFC.ST_XfcTouchProbeOptions;
  _XfcTriggerRef              : Tc2_MC2_XFC.XFC_TRIGGER_REF;
  _XfcTriggerRef_MT           : Tc2_MC2_XFC.XFC_MT_TRIGGER_REF;      // multi timestamping
  //_XfcEl1258Interface_MT      : Tc2_MC2_XFC.EL1258_MT_IoInterface;   // multi timestamping
  _XfcRecordedPosition_MT     : Tc2_MC2_XFC.ST_RecordedPosition;     // multi timestamping


  // outputs
  _XfcOutputEL2252            : Tc2_MC2_XFC.XFC_TouchProbe;
  _XfcOutputEL2258            : Tc2_MC2_XFC.XFC_EL2258_MultiEdge;

 
  // work vars

END_VAR

METHOD Check : BOOL
VAR_INST
  _idx        : UINT;
  _eCheck     : E_XFC_CHECK;
END_VAR

FOR _idx := 1 TO MAX_AXIS
DO
  IF NOT (_ItfAxis[_idx] <> 0)
  THEN
    _eCheck       := E_XFC_CHECK.XFC_CHECK_REF_AXIS_ITF;
    RETURN;
  END_IF
END_FOR




_eCheck           := E_XFC_CHECK.XFC_CHECK_DONE;
Check             := TRUE;
END_METHOD

//-----------------------------------------------------------------------------------------------------------
// GetIndex
//
// HAUD
// 18.07.2024
// - input:  TwinCAT NC Axis ID
// - output: index in AXIS_REF array
//-----------------------------------------------------------------------------------------------------------
METHOD GetIndex : UDINT
VAR_INPUT
  AxisId        : UDINT;
END_VAR
VAR
  _idx          : UDINT;
END_VAR

FOR _idx := 1 TO TO_UDINT(MAX_AXIS)
DO
  IF (_ItfAxis[_idx].AxisRef.NcToPlc.AxisId > 0)
  THEN
    IF (_ItfAxis[_idx].AxisRef.NcToPlc.AxisId = AxisId)
    THEN
      GetIndex      := _idx;
      RETURN;
    END_IF
  END_IF
END_FOR

GetIndex          := _idx;
END_METHOD

PROPERTY ItfAxis : ARRAY[1..MAX_AXIS]       OF I_McAxis
SET
_ItfAxis := ItfAxis;
END_SET
END_PROPERTY

METHOD PositionAtTime : E_PROGRESS
VAR_INPUT
  Execute         : BOOL;
  AxisId          : UDINT;                    // NC Axis ID
  DcTime          : Tc2_EtherCAT.T_DCTIME32;  // lower part Dctime of event
  MessageLevel    : E_MessageType := E_MessageType.eMessageError;  // switch for detailed logging if required
END_VAR
VAR_INST
  _eState         : E_PROGRESS;

  _stMsg          : ST_Message;
  _bError         : BOOL;
  _udiErrorId     : UDINT;
  _AxisIndex      : UDINT;
END_VAR
IF NOT Execute THEN _eState     := E_PROGRESS.PROGRESS_INIT;  END_IF
IF NOT Check() THEN PositionAtTime   := E_PROGRESS.PROGRESS_ERROR; END_IF

CASE _eState
OF
  E_PROGRESS.PROGRESS_INIT:
    IF Execute
    THEN
      _AxisIndex                := GetIndex(AxisId);
      _bError                   := FALSE;
      _udiErrorId               := 0;
      _eState                   := E_PROGRESS.PROGRESS_BUSY;

      IF (MessageLevel = E_MessageType.eMessageVerbose)
      THEN
        _stMsg.eType            := E_MessageType.eMessageVerbose;
        _stMsg.eDevice          := _eDeviceAxis;
        _stMsg.eSubdevice       := XfcPositionAtTime;
        _stMsg.iErrorNumber     := 0;
        _stMsg.sText            := TO_STRING(_eState);

        f_MessageSet(_stMsg);
      END_IF

      IF NOT (_AxisIndex > 0)
      THEN
        _stMsg.eType            := E_MessageType.eMessageError;
        _stMsg.eDevice          := _eDeviceAxis;
        _stMsg.eSubdevice       := XfcPositionAtTime;
        _stMsg.iErrorNumber     := _AxisIndex;
        _stMsg.sText            := TO_STRING(E_XFC_CHECK.XFC_CHECK_AXIS_INDEX);

        _bError                 := TRUE;
        _eState                 := E_PROGRESS.PROGRESS_STILL_WORKING;
      END_IF
    END_IF
END_CASE
//-----------------------------------------------------------------------------
//-----------------------------------------------------------------------------
CASE _eState
OF
  E_PROGRESS.PROGRESS_BUSY:
    _eState                     := E_PROGRESS.PROGRESS_STILL_WORKING;

    _XfcPositionAtTime[_AxisIndex](
                    DcTime      := DcTime, 
                    Options     := _XfcNcTimeConversionOptions[_AxisIndex], 
                    Position    => _XfcRecordedPosition[_AxisIndex], 
                    Error       => _bError, 
                    ErrorID     => _udiErrorId, 
                    Axis        := _ItfAxis[_AxisIndex].AxisRef);
END_CASE
//-----------------------------------------------------------------------------
//-----------------------------------------------------------------------------
CASE _eState
OF
  E_PROGRESS.PROGRESS_STILL_WORKING:
    IF NOT _bError
    THEN
      _eState                   := E_PROGRESS.PROGRESS_DONE;
      IF (MessageLevel > E_MessageType.eMessageWarning)
      THEN
        _stMsg.eType            := E_MessageType.eMessageInfo;
        _stMsg.eDevice          := _eDeviceAxis;
        _stMsg.eSubdevice       := XfcPositionAtTime;
        _stMsg.iErrorNumber     := 0;
        _stMsg.sText            := TO_STRING(_eState);

        f_MessageSet(_stMsg);
      END_IF
    ELSE
      _eState                   := E_PROGRESS.PROGRESS_ERROR;

      _stMsg.eType              := E_MessageType.eMessageError;
      _stMsg.eDevice            := _eDeviceAxis;
      _stMsg.eSubdevice         := XfcPositionAtTime;
      _stMsg.iErrorNumber       := _udiErrorId;
      _stMsg.sText              := TO_STRING(_eState);

      f_MessageSet(_stMsg);
    END_IF
END_CASE



PositionAtTime                  := _eState;
END_METHOD

METHOD TimeOfPosition : E_PROGRESS
VAR_INPUT
  Execute         : BOOL;
  AxisId          : UDINT;                    // NC Axis ID
  Position        : LREAL;
  MessageLevel    : E_MessageType := E_MessageType.eMessageError;  // switch for detailed logging if required
END_VAR
VAR_INST
  _eState         : E_PROGRESS;

  _stMsg          : ST_Message;
  _bError         : BOOL;
  _udiErrorId     : UDINT;
  _AxisIndex      : UDINT;
END_VAR
IF NOT Execute THEN _eState     := E_PROGRESS.PROGRESS_INIT;  END_IF
IF NOT Check() THEN TimeOfPosition   := E_PROGRESS.PROGRESS_ERROR; END_IF

CASE _eState
OF
  E_PROGRESS.PROGRESS_INIT:
    IF Execute
    THEN
      _AxisIndex                := GetIndex(AxisId);
      _bError                   := FALSE;
      _udiErrorId               := 0;
      _eState                   := E_PROGRESS.PROGRESS_BUSY;

      IF (MessageLevel = E_MessageType.eMessageVerbose)
      THEN
        _stMsg.eType            := E_MessageType.eMessageVerbose;
        _stMsg.eDevice          := _eDeviceAxis;
        _stMsg.eSubdevice       := XfcTimeOfPosition;
        _stMsg.iErrorNumber     := 0;
        _stMsg.sText            := TO_STRING(_eState);

        f_MessageSet(_stMsg);
      END_IF

      IF NOT (_AxisIndex > 0)
      THEN
        _stMsg.eType            := E_MessageType.eMessageError;
        _stMsg.eDevice          := _eDeviceAxis;
        _stMsg.eSubdevice       := XfcTimeOfPosition;
        _stMsg.iErrorNumber     := _AxisIndex;
        _stMsg.sText            := TO_STRING(E_XFC_CHECK.XFC_CHECK_AXIS_INDEX);

        _bError                 := TRUE;
        _eState                 := E_PROGRESS.PROGRESS_STILL_WORKING;
      END_IF
    END_IF
END_CASE
//-----------------------------------------------------------------------------
//-----------------------------------------------------------------------------
CASE _eState
OF
  E_PROGRESS.PROGRESS_BUSY:
    _eState                     := E_PROGRESS.PROGRESS_STILL_WORKING;

    _XfcTimeOfPosition[_AxisIndex](
	                  Position    := Position, 
                    Options     := _XfcNcTimeConversionOptions[_AxisIndex], 
                    DcTime      => _XfcRecordedTime[_AxisIndex], 
                    Error       => _bError, 
                    ErrorID     => _udiErrorId, 
                    Axis        := _ItfAxis[_AxisIndex].AxisRef);
END_CASE
//-----------------------------------------------------------------------------
//-----------------------------------------------------------------------------
CASE _eState
OF
  E_PROGRESS.PROGRESS_STILL_WORKING:
    IF NOT _bError
    THEN
      _eState                   := E_PROGRESS.PROGRESS_DONE;
      IF (MessageLevel > E_MessageType.eMessageWarning)
      THEN
        _stMsg.eType            := E_MessageType.eMessageInfo;
        _stMsg.eDevice          := _eDeviceAxis;
        _stMsg.eSubdevice       := XfcTimeOfPosition;
        _stMsg.iErrorNumber     := 0;
        _stMsg.sText            := TO_STRING(_eState);

        f_MessageSet(_stMsg);
      END_IF
    ELSE
      _eState                   := E_PROGRESS.PROGRESS_ERROR;

      _stMsg.eType              := E_MessageType.eMessageError;
      _stMsg.eDevice            := _eDeviceAxis;
      _stMsg.eSubdevice         := XfcTimeOfPosition;
      _stMsg.iErrorNumber       := _udiErrorId;
      _stMsg.sText              := TO_STRING(_eState);

      f_MessageSet(_stMsg);
    END_IF
END_CASE



TimeOfPosition                  := _eState;
END_METHOD

METHOD TimeToPosition : E_PROGRESS
VAR_INPUT
  Execute         : BOOL;
  AxisId          : UDINT;                    // NC Axis ID
  TargetPosition  : LREAL;
  MessageLevel    : E_MessageType := E_MessageType.eMessageError;  // switch for detailed logging if required
END_VAR
VAR_INST
  _eState         : E_PROGRESS;

  _stMsg          : ST_Message;
  _bError         : BOOL;
  _udiErrorId     : UDINT;
  _AxisIndex      : UDINT;
END_VAR
IF NOT Execute THEN _eState     := E_PROGRESS.PROGRESS_INIT;  END_IF
IF NOT Check() THEN TimeToPosition   := E_PROGRESS.PROGRESS_ERROR; END_IF

CASE _eState
OF
  E_PROGRESS.PROGRESS_INIT:
    IF Execute
    THEN
      _AxisIndex                := GetIndex(AxisId);
      _bError                   := FALSE;
      _udiErrorId               := 0;
      _eState                   := E_PROGRESS.PROGRESS_BUSY;

      IF (MessageLevel = E_MessageType.eMessageVerbose)
      THEN
        _stMsg.eType            := E_MessageType.eMessageVerbose;
        _stMsg.eDevice          := _eDeviceAxis;
        _stMsg.eSubdevice       := XfcTimeToPosition;
        _stMsg.iErrorNumber     := 0;
        _stMsg.sText            := TO_STRING(_eState);

        f_MessageSet(_stMsg);
      END_IF

      IF NOT (_AxisIndex > 0)
      THEN
        _stMsg.eType            := E_MessageType.eMessageError;
        _stMsg.eDevice          := _eDeviceAxis;
        _stMsg.eSubdevice       := XfcTimeToPosition;
        _stMsg.iErrorNumber     := _AxisIndex;
        _stMsg.sText            := TO_STRING(E_XFC_CHECK.XFC_CHECK_AXIS_INDEX);

        _bError                 := TRUE;
        _eState                 := E_PROGRESS.PROGRESS_STILL_WORKING;
      END_IF
    END_IF
END_CASE
//-----------------------------------------------------------------------------
//-----------------------------------------------------------------------------
CASE _eState
OF
  E_PROGRESS.PROGRESS_BUSY:
    _eState                     := E_PROGRESS.PROGRESS_STILL_WORKING;

    _XfcTimeToPosition[_AxisIndex](
                Position        := TargetPosition, 
                Options         := _XfcNcTimeConversionOptions[_AxisIndex], 
                Duration        => _XfcDurationToPosition[_AxisIndex], 
                TimeOfPosition  => _XfcDcTimeOfPosition[_AxisIndex], 
                Error           => _bError, 
                ErrorID         => _udiErrorId, 
                Axis            := _ItfAxis[_AxisIndex].AxisRef);
END_CASE
//-----------------------------------------------------------------------------
//-----------------------------------------------------------------------------
CASE _eState
OF
  E_PROGRESS.PROGRESS_STILL_WORKING:
    IF NOT _bError
    THEN
      _eState                   := E_PROGRESS.PROGRESS_DONE;
      IF (MessageLevel > E_MessageType.eMessageWarning)
      THEN
        _stMsg.eType            := E_MessageType.eMessageInfo;
        _stMsg.eDevice          := _eDeviceAxis;
        _stMsg.eSubdevice       := XfcTimeToPosition;
        _stMsg.iErrorNumber     := 0;
        _stMsg.sText            := TO_STRING(_eState);

        f_MessageSet(_stMsg);
      END_IF
    ELSE
      _eState                   := E_PROGRESS.PROGRESS_ERROR;

      _stMsg.eType              := E_MessageType.eMessageError;
      _stMsg.eDevice            := _eDeviceAxis;
      _stMsg.eSubdevice         := XfcTimeToPosition;
      _stMsg.iErrorNumber       := _udiErrorId;
      _stMsg.sText              := TO_STRING(_eState);

      f_MessageSet(_stMsg);
    END_IF
END_CASE



TimeToPosition                  := _eState;
END_METHOD

METHOD TimeToPositionModulo : E_PROGRESS
VAR_INPUT
  Execute         : BOOL;
  AxisId          : UDINT;                    // NC Axis ID
  ModuloPosition  : LREAL;
  ModuloFactor    : LREAL;
  MessageLevel    : E_MessageType := E_MessageType.eMessageError;  // switch for detailed logging if required
END_VAR
VAR_INST
  _eState         : E_PROGRESS;

  _stMsg          : ST_Message;
  _bError         : BOOL;
  _udiErrorId     : UDINT;
  _AxisIndex      : UDINT;
END_VAR
IF NOT Execute THEN _eState     := E_PROGRESS.PROGRESS_INIT;  END_IF
IF NOT Check() THEN TimeToPositionModulo   := E_PROGRESS.PROGRESS_ERROR; END_IF

CASE _eState
OF
  E_PROGRESS.PROGRESS_INIT:
    IF Execute
    THEN
      _AxisIndex                := GetIndex(AxisId);
      _bError                   := FALSE;
      _udiErrorId               := 0;
      _eState                   := E_PROGRESS.PROGRESS_BUSY;

      IF (MessageLevel = E_MessageType.eMessageVerbose)
      THEN
        _stMsg.eType            := E_MessageType.eMessageVerbose;
        _stMsg.eDevice          := _eDeviceAxis;
        _stMsg.eSubdevice       := XfcTimeToModuloPosition;
        _stMsg.iErrorNumber     := 0;
        _stMsg.sText            := TO_STRING(_eState);

        f_MessageSet(_stMsg);
      END_IF

      IF NOT (_AxisIndex > 0)
      THEN
        _stMsg.eType            := E_MessageType.eMessageError;
        _stMsg.eDevice          := _eDeviceAxis;
        _stMsg.eSubdevice       := XfcTimeToModuloPosition;
        _stMsg.iErrorNumber     := _AxisIndex;
        _stMsg.sText            := TO_STRING(E_XFC_CHECK.XFC_CHECK_AXIS_INDEX);

        _bError                 := TRUE;
        _eState                 := E_PROGRESS.PROGRESS_STILL_WORKING;
      END_IF
    END_IF
END_CASE
//-----------------------------------------------------------------------------
//-----------------------------------------------------------------------------
CASE _eState
OF
  E_PROGRESS.PROGRESS_BUSY:
    _eState                     := E_PROGRESS.PROGRESS_STILL_WORKING;

    _XfcTimeToModuloPosition[_AxisIndex](
                Position        := ModuloPosition, 
                ModuloFactor    := ModuloFactor, 
                Options         := _XfcNcTimeConversionOptions[_AxisIndex], 
                Duration        => _XfcDurationToPosition[_AxisIndex], 
                AbsolutePosition=> _XfcRecordedPosition[_AxisIndex], 
                TimeOfPosition  => _XfcDcTimeOfPosition[_AxisIndex], 
                Error           => _bError, 
                ErrorID         => _udiErrorId, 
                Axis            := _ItfAxis[_AxisIndex].AxisRef);
END_CASE
//-----------------------------------------------------------------------------
//-----------------------------------------------------------------------------
CASE _eState
OF
  E_PROGRESS.PROGRESS_STILL_WORKING:
    IF NOT _bError
    THEN
      _eState                   := E_PROGRESS.PROGRESS_DONE;
      IF (MessageLevel > E_MessageType.eMessageWarning)
      THEN
        _stMsg.eType            := E_MessageType.eMessageInfo;
        _stMsg.eDevice          := _eDeviceAxis;
        _stMsg.eSubdevice       := XfcTimeToModuloPosition;
        _stMsg.iErrorNumber     := 0;
        _stMsg.sText            := TO_STRING(_eState);

        f_MessageSet(_stMsg);
      END_IF
    ELSE
      _eState                   := E_PROGRESS.PROGRESS_ERROR;

      _stMsg.eType              := E_MessageType.eMessageError;
      _stMsg.eDevice            := _eDeviceAxis;
      _stMsg.eSubdevice         := XfcTimeToModuloPosition;
      _stMsg.iErrorNumber       := _udiErrorId;
      _stMsg.sText              := TO_STRING(_eState);

      f_MessageSet(_stMsg);
    END_IF
END_CASE

TimeToPositionModulo                  := _eState;
END_METHOD

METHOD WaitForPosition : E_PROGRESS
VAR_INPUT
  Execute         : BOOL;
  AxisId          : UDINT;                    // NC Axis ID
  TargetPosition  : LREAL;
  MessageLevel    : E_MessageType := E_MessageType.eMessageError;  // switch for detailed logging if required
END_VAR
VAR_INST
  _eState         : E_PROGRESS;

  _stMsg          : ST_Message;
  _bError         : BOOL;
  _udiErrorId     : UDINT;
  _AxisIndex      : UDINT;
END_VAR
IF NOT Execute THEN _eState     := E_PROGRESS.PROGRESS_INIT;  END_IF
IF NOT Check() THEN WaitForPosition   := E_PROGRESS.PROGRESS_ERROR; END_IF

CASE _eState
OF
  E_PROGRESS.PROGRESS_INIT:
    IF Execute
    THEN
      _AxisIndex                := GetIndex(AxisId);
      _bError                   := FALSE;
      _udiErrorId               := 0;
      _eState                   := E_PROGRESS.PROGRESS_BUSY;

      IF (MessageLevel = E_MessageType.eMessageVerbose)
      THEN
        _stMsg.eType            := E_MessageType.eMessageVerbose;
        _stMsg.eDevice          := _eDeviceAxis;
        _stMsg.eSubdevice       := XfcWaitForPosition;
        _stMsg.iErrorNumber     := 0;
        _stMsg.sText            := TO_STRING(_eState);

        f_MessageSet(_stMsg);
      END_IF

      IF NOT (_AxisIndex > 0)
      THEN
        _stMsg.eType            := E_MessageType.eMessageError;
        _stMsg.eDevice          := _eDeviceAxis;
        _stMsg.eSubdevice       := XfcWaitForPosition;
        _stMsg.iErrorNumber     := _AxisIndex;
        _stMsg.sText            := TO_STRING(E_XFC_CHECK.XFC_CHECK_AXIS_INDEX);

        _bError                 := TRUE;
        _eState                 := E_PROGRESS.PROGRESS_STILL_WORKING;
      END_IF
    END_IF
END_CASE
//-----------------------------------------------------------------------------
//-----------------------------------------------------------------------------
CASE _eState
OF
  E_PROGRESS.PROGRESS_BUSY:
    _eState                     := E_PROGRESS.PROGRESS_PREPARE;

    _XfcTimeToPosition[_AxisIndex](
                Position        := TargetPosition, 
                Options         := _XfcNcTimeConversionOptions[_AxisIndex], 
                Duration        => _XfcDurationToPosition[_AxisIndex], 
                TimeOfPosition  => , 
                Error           => _bError, 
                ErrorID         => _udiErrorId, 
                Axis            := _ItfAxis[_AxisIndex].AxisRef);

END_CASE
//-----------------------------------------------------------------------------
//-----------------------------------------------------------------------------
CASE _eState
OF
  E_PROGRESS.PROGRESS_PREPARE:

    IF NOT _bError
    THEN
      IF (_XfcTimeToPosition[_AxisIndex].Duration < 10_000_000)
      THEN
        _eState                 := E_PROGRESS.PROGRESS_STILL_WORKING;
      ELSE
        _eState                 := E_PROGRESS.PROGRESS_BUSY;
      END_IF
    ELSE
      IF (_udiErrorId <> 17250)
      THEN
        // axis is not yet in range --> retry
        _eState                 := E_PROGRESS.PROGRESS_BUSY;
      ELSE
        // position will not be reachable --> error
        _eState                 := E_PROGRESS.PROGRESS_STILL_WORKING;  
      END_IF
    END_IF
END_CASE
//-----------------------------------------------------------------------------
//-----------------------------------------------------------------------------
CASE _eState
OF
  E_PROGRESS.PROGRESS_STILL_WORKING:
    IF NOT _bError
    THEN
      _eState                   := E_PROGRESS.PROGRESS_DONE;
      IF (MessageLevel > E_MessageType.eMessageWarning)
      THEN
        _stMsg.eType            := E_MessageType.eMessageInfo;
        _stMsg.eDevice          := _eDeviceAxis;
        _stMsg.eSubdevice       := XfcWaitForPosition;
        _stMsg.iErrorNumber     := TO_ULINT(_XfcDurationToPosition[_AxisIndex]);
        _stMsg.sText            := TO_STRING(_eState);

        f_MessageSet(_stMsg);
      END_IF
    ELSE
      _eState                   := E_PROGRESS.PROGRESS_ERROR;

      _stMsg.eType              := E_MessageType.eMessageError;
      _stMsg.eDevice            := _eDeviceAxis;
      _stMsg.eSubdevice         := XfcWaitForPosition;
      _stMsg.iErrorNumber       := _udiErrorId;
      _stMsg.sText              := TO_STRING(_eState);

      f_MessageSet(_stMsg);
    END_IF
END_CASE


WaitForPosition                 := _eState;
END_METHOD

END_FUNCTION_BLOCK

// ---- FUNCTIONS/TOUCH_PROBE/FB_TouchProbe.TcPOU
FUNCTION_BLOCK FB_TouchProbe EXTENDS FB_Xfc
VAR
  _Ctrl             : REFERENCE TO ARRAY[1..MAX_TOUCH_PROBE] OF ST_CTRL_TOUCH_PROBE;
  _State            : REFERENCE TO ARRAY[1..MAX_TOUCH_PROBE] OF ST_STATE_TOUCH_PROBE;

  _Input            : POINTER TO ARRAY[1..MAX_TOUCH_PROBE] OF ST_MTI_Input;
  _InputState       : POINTER TO ARRAY[1..MAX_TOUCH_PROBE] OF ST_MTI_STATUS;

  _Index            : UDINT;
  _AxisId           : UDINT;
  _AxisIndex        : UDINT;

  _CtrlLocal        : ST_CTRL_TOUCH_PROBE;  // control data is copied to local on start of function
  _McDirection      : Tc2_MC2.MC_Direction;

  _eStateProgress   : E_PROGRESS;
  _eResult          : E_PROGRESS;

  _rtrigEnable      : Tc2_Standard.R_TRIG;
  _TrigCount        : UDINT;

  _CurrentTime      : ULINT;
  _CurrentTimeShort : UDINT;
  _LatchTime        : UDINT;
  _LatchState       : Bool;

  _bError           : BOOL;
  _stMsg            : ST_Message;
  _MessageLevel     : E_MessageType;
END_VAR

PROPERTY Ctrl : REFERENCE TO ARRAY [1..MAX_TOUCH_PROBE] OF ST_CTRL_TOUCH_PROBE
SET
_Ctrl REF= Ctrl;
END_SET
END_PROPERTY

METHOD Cycle : BOOL
VAR_INPUT
END_VAR
//-----------------------------------------------------------------------------
//-----------------------------------------------------------------------------
//  Check Enable
//-----------------------------------------------------------------------------
IF NOT _Ctrl[_Index].Enable
THEN
  // clear function state if not enabled
  _eStateProgress                   := E_PROGRESS.PROGRESS_INVALID;
  _LatchState                       := FALSE;
  _State[_Index].State              := TO_UINT(_eStateProgress);
END_IF
//-----------------------------------------------------------------------------
//-----------------------------------------------------------------------------
//  set message device
//-----------------------------------------------------------------------------
_eDeviceFunction                    := e_Device.XfcTouchProbe + _Index;
//-----------------------------------------------------------------------------
//-----------------------------------------------------------------------------
//  rising trigger react to enable command
//-----------------------------------------------------------------------------
_rtrigEnable(CLK                    := _Ctrl[_Index].Enable);
//-----------------------------------------------------------------------------
//-----------------------------------------------------------------------------
//  main state machine
//-----------------------------------------------------------------------------
CASE _eStateProgress
OF
  E_PROGRESS.PROGRESS_INVALID:      // check input data
    IF _rtrigEnable.Q
    THEN
      _State[_Index].State          := TO_UINT(E_PROGRESS.PROGRESS_BUSY);
      _State[_Index].LatchPositive  := 0.0;
      _State[_Index].LatchNegative  := 0.0;

      _bError                       := FALSE;
      _eStateProgress               := E_PROGRESS.PROGRESS_INIT;

      _CtrlLocal                    := _Ctrl[_Index];   // copy control data to local, you may write new data onto struct as long as .Enable stays TRUE
      _CurrentTime                  := Tc2_EtherCAT.F_GetCurDcTickTime64();
      _CurrentTimeShort             := TO_UDINT(_CurrentTime AND 16#FFFFFFFF);

      _AxisId                       := _CtrlLocal.AxisId;   // TwinCAT NC AxisId
      _AxisIndex                    := GetIndex(_AxisId);   // corresponding index in axis array

      _stMsg.iErrorNumber           := 0;

      IF NOT (_AxisIndex > 0) OR NOT (_AxisId > 0)
      THEN
        _bError                     := TRUE;
        _stMsg.iErrorNumber         := 1;
        _stMsg.sText                := 'AxisId Invalid ';
        _eStateProgress             := E_PROGRESS.PROGRESS_STILL_WORKING;
      END_IF

      IF NOT (_CtrlLocal.Direction = MC_Positive_Direction) OR 
         NOT (_CtrlLocal.Direction = MC_Negative_Direction)
      THEN
        _bError                     := TRUE;
        _stMsg.iErrorNumber         := 2;
        _stMsg.sText                := 'Direction Invalid ';
        _eStateProgress             := E_PROGRESS.PROGRESS_STILL_WORKING;
      END_IF

      IF NOT IsFinite(F_LReal(_CtrlLocal.PositionStart))
      THEN
        _bError                     := TRUE;
        _stMsg.iErrorNumber         := 3;
        _stMsg.sText                := 'PositionStart not finite ';
        _eStateProgress             := E_PROGRESS.PROGRESS_STILL_WORKING;
      END_IF

      IF NOT IsFinite(F_LReal(_CtrlLocal.PositionEnd))
      THEN
        _bError                     := TRUE;
        _stMsg.iErrorNumber         := 4;
        _stMsg.sText                := 'PositionEnd not finite ';
        _eStateProgress             := E_PROGRESS.PROGRESS_STILL_WORKING;
      END_IF
    END_IF

  E_PROGRESS.PROGRESS_INIT:
      _eDeviceAxis                  := e_Device.XfcAxis + (_CtrlLocal.AxisId);
      _eStateProgress               := E_PROGRESS.PROGRESS_BUSY;

      IF (_MessageLevel = E_MessageType.eMessageVerbose)
      THEN
        _stMsg.eType                := E_MessageType.eMessageVerbose;
        _stMsg.eDevice              := _eDeviceFunction;
        _stMsg.eSubdevice           := e_Subdevice.XfcTouchProbe;
        _stMsg.iErrorNumber         := _eDeviceAxis;
        _stMsg.sText                := concat(TO_STRING(_eStateProgress), ': ');
        _stMsg.sText                := concat(_stMsg.sText, TO_STRING(e_Device.XfcAxis));
        _stMsg.sText                := concat(_stMsg.sText, '_ID_');
        _stMsg.sText                := concat(_stMsg.sText, TO_STRING(_AxisId));

        f_MessageSet(_stMsg);
      END_IF
END_CASE
//-----------------------------------------------------------------------------
//-----------------------------------------------------------------------------
CASE _eStateProgress
OF
  E_PROGRESS.PROGRESS_BUSY:
    _McDirection                    := _CtrlLocal.Direction;
    CASE _McDirection
    OF
      MC_Positive_Direction:
        IF (_ItfAxis[_AxisIndex].Position >= _CtrlLocal.PositionStart)
        THEN
          _eResult                  := PositionAtTime(FALSE, _CtrlLocal.AxisId, 0, _MessageLevel);
          _eStateProgress           := E_PROGRESS.PROGRESS_PREPARE;
        END_IF

      MC_Negative_Direction:
        IF (_ItfAxis[_AxisIndex].Position <= _CtrlLocal.PositionStart)
        THEN
          _eResult                  := PositionAtTime(FALSE, _CtrlLocal.AxisId, 0, _MessageLevel);
          _eStateProgress           := E_PROGRESS.PROGRESS_PREPARE;
        END_IF
    END_CASE
END_CASE
//-----------------------------------------------------------------------------
//-----------------------------------------------------------------------------
CASE _eStateProgress
OF
  E_PROGRESS.PROGRESS_PREPARE:
    CASE _McDirection
    OF
      MC_Positive_Direction:
        IF (_ItfAxis[_AxisIndex].Position > _CtrlLocal.PositionEnd)
        THEN
          _bError                   := TRUE;
          _stMsg.iErrorNumber       := 5;
          _stMsg.sText              := 'PositionEnd reached, no rising trigger ';
          _eStateProgress           := E_PROGRESS.PROGRESS_STILL_WORKING;
    
        ELSIF (_Input^[_Index].EventState) OR
              (_Input^[_Index].EventTime > _CurrentTimeShort)
        THEN
          _LatchState               := _Input^[_Index].EventState;
          _LatchTime                := _Input^[_Index].EventTime;
    
          IF (_MessageLevel = E_MessageType.eMessageVerbose)
          THEN
            _stMsg.eType            := E_MessageType.eMessageVerbose;
            _stMsg.eDevice          := _eDeviceFunction;
            _stMsg.eSubdevice       := e_Subdevice.XfcTouchProbe;
            _stMsg.iErrorNumber     := _LatchTime;
            _stMsg.sText            := concat(TO_STRING(_eStateProgress), ': ');
            _stMsg.sText            := concat(_stMsg.sText, TO_STRING(e_Device.XfcAxis));
    
            f_MessageSet(_stMsg);
          END_IF
          _eStateProgress           := E_PROGRESS.PROGRESS_STARTUP;
        END_IF

      MC_Negative_Direction:
        IF (_ItfAxis[_AxisIndex].Position < _CtrlLocal.PositionEnd)
        THEN
          _bError                   := TRUE;
          _stMsg.iErrorNumber       := 5;
          _stMsg.sText              := 'PositionEnd reached, no rising trigger ';
          _eStateProgress           := E_PROGRESS.PROGRESS_STILL_WORKING;
    
        ELSIF (_Input^[_Index].EventState) OR
              (_Input^[_Index].EventTime > _CurrentTimeShort)
        THEN
          _LatchState               := _Input^[_Index].EventState;
          _LatchTime                := _Input^[_Index].EventTime;
    
          IF (_MessageLevel = E_MessageType.eMessageVerbose)
          THEN
            _stMsg.eType            := E_MessageType.eMessageVerbose;
            _stMsg.eDevice          := _eDeviceFunction;
            _stMsg.eSubdevice       := e_Subdevice.XfcTouchProbe;
            _stMsg.iErrorNumber     := _LatchTime;
            _stMsg.sText            := concat(TO_STRING(_eStateProgress), ': ');
            _stMsg.sText            := concat(_stMsg.sText, TO_STRING(e_Device.XfcAxis));
    
            f_MessageSet(_stMsg);
          END_IF
          _eStateProgress           := E_PROGRESS.PROGRESS_STARTUP;
        END_IF
    END_CASE
END_CASE
//-----------------------------------------------------------------------------
//-----------------------------------------------------------------------------
CASE _eStateProgress
OF
  E_PROGRESS.PROGRESS_STARTUP:
    _eResult                        := PositionAtTime(TRUE, _CtrlLocal.AxisId, _LatchTime, _MessageLevel);

    IF (_eResult = E_PROGRESS.PROGRESS_ERROR)
    THEN
      _bError                       := TRUE;
      _stMsg.iErrorNumber           := 7;
      _stMsg.sText                  := 'PositionAtTime LatchPositive ';
      _eStateProgress               := E_PROGRESS.PROGRESS_STILL_WORKING;
      _eResult                      := PositionAtTime(FALSE, _CtrlLocal.AxisId, 0, _MessageLevel);

    ELSIF (_eResult = E_PROGRESS.PROGRESS_DONE)
    THEN
      _State[_Index].LatchPositive  := _XfcRecordedPosition[_AxisIndex];

      _CurrentTime                  := Tc2_EtherCAT.F_GetCurDcTickTime64();
      _CurrentTimeShort             := TO_UDINT(_CurrentTime AND 16#FFFFFFFF);

      IF (_MessageLevel = E_MessageType.eMessageVerbose)
      THEN
        _stMsg.eType                := E_MessageType.eMessageVerbose;
        _stMsg.eDevice              := _eDeviceFunction;
        _stMsg.eSubdevice           := e_Subdevice.XfcTouchProbe;
        _stMsg.iErrorNumber         := _LatchTime;
        _stMsg.sText                := concat(TO_STRING(_eStateProgress), ': ');
        _stMsg.sText                := concat(_stMsg.sText, TO_STRING(_XfcRecordedPosition[_AxisIndex]));

        f_MessageSet(_stMsg);
      END_IF
      _eStateProgress               := E_PROGRESS.PROGRESS_CHECK;
      _eResult                      := PositionAtTime(FALSE, _CtrlLocal.AxisId, 0, _MessageLevel);
    END_IF
END_CASE
//-----------------------------------------------------------------------------
//-----------------------------------------------------------------------------
CASE _eStateProgress
OF
  E_PROGRESS.PROGRESS_CHECK:
    CASE _McDirection
    OF
      MC_Positive_Direction:
        IF (_ItfAxis[_AxisIndex].Position > _CtrlLocal.PositionEnd)
        THEN
          _bError                   := TRUE;
          _stMsg.iErrorNumber       := 6;
          _stMsg.sText              := concat('PositionEnd reached, no falling trigger :', TO_STRING(_ItfAxis[_AxisIndex].Position));
          _eStateProgress           := E_PROGRESS.PROGRESS_STILL_WORKING;
    
        ELSIF NOT (_Input^[_Index].EventState) OR
              (_Input^[_Index].EventTime > _LatchTime - 1_000)
        THEN
          _LatchState               := _Input^[_Index].EventState;
          _LatchTime                := _Input^[_Index].EventTime;
    
          IF (_MessageLevel = E_MessageType.eMessageVerbose)
          THEN
            _stMsg.eType            := E_MessageType.eMessageVerbose;
            _stMsg.eDevice          := _eDeviceFunction;
            _stMsg.eSubdevice       := e_Subdevice.XfcTouchProbe;
            _stMsg.iErrorNumber     := _LatchTime;
            _stMsg.sText            := concat(TO_STRING(_eStateProgress), ': ');
            _stMsg.sText            := concat(_stMsg.sText, TO_STRING(e_Device.XfcAxis));
    
            f_MessageSet(_stMsg);
          END_IF
          _eStateProgress           := E_PROGRESS.PROGRESS_OCCUPIED;
        END_IF

      MC_Negative_Direction:
        IF (_ItfAxis[_AxisIndex].Position < _CtrlLocal.PositionEnd)
        THEN
          _bError                   := TRUE;
          _stMsg.iErrorNumber       := 6;
          _stMsg.sText              := concat('PositionEnd reached, no falling trigger :', TO_STRING(_ItfAxis[_AxisIndex].Position));
          _eStateProgress           := E_PROGRESS.PROGRESS_STILL_WORKING;
    
        ELSIF NOT (_Input^[_Index].EventState) OR
              (_Input^[_Index].EventTime > _LatchTime - 1_000)
        THEN
          _LatchState               := _Input^[_Index].EventState;
          _LatchTime                := _Input^[_Index].EventTime;
    
          IF (_MessageLevel = E_MessageType.eMessageVerbose)
          THEN
            _stMsg.eType            := E_MessageType.eMessageVerbose;
            _stMsg.eDevice          := _eDeviceFunction;
            _stMsg.eSubdevice       := e_Subdevice.XfcTouchProbe;
            _stMsg.iErrorNumber     := _LatchTime;
            _stMsg.sText            := concat(TO_STRING(_eStateProgress), ': ');
            _stMsg.sText            := concat(_stMsg.sText, TO_STRING(e_Device.XfcAxis));
    
            f_MessageSet(_stMsg);
          END_IF
          _eStateProgress           := E_PROGRESS.PROGRESS_OCCUPIED;
        END_IF
    END_CASE
END_CASE
//-----------------------------------------------------------------------------
//-----------------------------------------------------------------------------
CASE _eStateProgress
OF
  E_PROGRESS.PROGRESS_OCCUPIED:
    _eResult                        := PositionAtTime(TRUE, _CtrlLocal.AxisId, _LatchTime, _MessageLevel);

    IF (_eResult = E_PROGRESS.PROGRESS_ERROR)
    THEN
      _bError                       := TRUE;
      _stMsg.iErrorNumber           := 8;
      _stMsg.sText                  := 'PositionAtTime LatchNegative: ';
      _eStateProgress               := E_PROGRESS.PROGRESS_STILL_WORKING;
      _eResult                      := PositionAtTime(FALSE, _CtrlLocal.AxisId, 0, _MessageLevel);

    ELSIF (_eResult = E_PROGRESS.PROGRESS_DONE)
    THEN
      _State[_Index].LatchNegative  := _XfcRecordedPosition[_AxisIndex];

      IF (_MessageLevel = E_MessageType.eMessageVerbose)
      THEN
        _stMsg.eType                := E_MessageType.eMessageVerbose;
        _stMsg.eDevice              := _eDeviceFunction;
        _stMsg.eSubdevice           := e_Subdevice.XfcTouchProbe;
        _stMsg.iErrorNumber         := _LatchTime;
        _stMsg.sText                := concat(TO_STRING(_eStateProgress), ': ');
        _stMsg.sText                := concat(_stMsg.sText, TO_STRING(_XfcRecordedPosition[_AxisIndex]));

        f_MessageSet(_stMsg);
      END_IF
      _eStateProgress               := E_PROGRESS.PROGRESS_WORKING;
      _eResult                      := PositionAtTime(FALSE, _CtrlLocal.AxisId, 0, _MessageLevel);
    END_IF
END_CASE
//-----------------------------------------------------------------------------
//-----------------------------------------------------------------------------
CASE _eStateProgress
OF
  E_PROGRESS.PROGRESS_WORKING:
    _eStateProgress                 := E_PROGRESS.PROGRESS_STILL_WORKING;
END_CASE
//-----------------------------------------------------------------------------
//-----------------------------------------------------------------------------
CASE _eStateProgress
OF
  E_PROGRESS.PROGRESS_STILL_WORKING:
    IF NOT _bError
    THEN
      _eStateProgress               := E_PROGRESS.PROGRESS_DONE;

      IF (_MessageLevel > E_MessageType.eMessageWarning)
      THEN
        _stMsg.eType                := E_MessageType.eMessageInfo;
        _stMsg.eDevice              := _eDeviceFunction;
        _stMsg.eSubdevice           := e_Subdevice.XfcTouchProbe;
        _stMsg.iErrorNumber         := _eDeviceAxis;
        _stMsg.sText                := concat(TO_STRING(_eStateProgress), ': ');
        _stMsg.sText                := concat(_stMsg.sText, TO_STRING(e_Device.XfcAxis));
        _stMsg.sText                := concat(_stMsg.sText, '_ID_');
        _stMsg.sText                := concat(_stMsg.sText, TO_STRING(_AxisId));

        f_MessageSet(_stMsg);
      END_IF
      _State[_Index].State          := TO_UINT(_eStateProgress);
    ELSE
      _eStateProgress               := E_PROGRESS.PROGRESS_ERROR;

      _stMsg.eType                  := E_MessageType.eMessageError;
      _stMsg.eDevice                := _eDeviceFunction;
      _stMsg.eSubdevice             := e_Subdevice.XfcTouchProbe;
      _stMsg.sText                  := concat(_stMsg.sText, TO_STRING(_eStateProgress));
      _stMsg.sText                  := concat(_stMsg.sText, ': ');
      _stMsg.sText                  := concat(_stMsg.sText, TO_STRING(e_Device.XfcAxis));
      _stMsg.sText                  := concat(_stMsg.sText, '_ID_');
      _stMsg.sText                  := concat(_stMsg.sText, TO_STRING(_AxisId));

      f_MessageSet(_stMsg);
      _State[_Index].State          := TO_UINT(_eStateProgress) + TO_UINT(_stMsg.iErrorNumber);
    END_IF
END_CASE
END_METHOD

PROPERTY Index : udint
GET
Index := _Index;
END_GET
SET
_Index := Index;
END_SET
END_PROPERTY

PROPERTY Input : pointer TO ARRAY [1..MAX_TOUCH_PROBE] OF ST_MTI_Input
SET
_Input := Input;
END_SET
END_PROPERTY

PROPERTY InputState : pointer TO ARRAY [1..MAX_TOUCH_PROBE] OF ST_MTI_STATUS
SET
_InputState := InputState;
END_SET
END_PROPERTY

PROPERTY MessageLevel : e_messagetype
GET
MessageLevel := _MessageLevel;
END_GET
SET
_MessageLevel := MessageLevel;
END_SET
END_PROPERTY

PROPERTY State :  REFERENCE TO ARRAY[1..MAX_TOUCH_PROBE] OF ST_STATE_TOUCH_PROBE;
SET
_State REF= State;
END_SET
END_PROPERTY

END_FUNCTION_BLOCK

// ---- NCI/FB_NciChannel.TcPOU
FUNCTION_BLOCK abstract FB_NciChannel IMPLEMENTS I_NciChannel
VAR
  ChannelDevice         : e_Device := e_Device.NciChannel;

// 2nd result of Check()
  _eCheck               : E_CHECK_STATE;

  _MessageLevel         : E_MessageType;

//NCI-Channel reference
  _NciChannelRef        : POINTER TO ST_NciChannel_Ref;

//Configured Group Axes
  _stCfgAxes            : POINTER TO ST_3D_Group;

//NCI-Group
  _fbBuildGroup         : Tc2_NCI.CfgBuildExt3DGroup;
  _fbClearGroup         : Tc2_NCI.CfgReconfigGroup;

  _fOverride            : LREAL := 100;

  _mdx,
  _adx                  : UINT;
  
//NCI-Program
{IF defined (WIN)}
  _sProg                : STRING(255) := 'C:\TwinCAT\Mc\Nci\Test_GST.nc';
{ELSE}
  _sProg                : STRING(255) := '/usr/local/etc/TwinCAT/Mc/Nci/Test_GST.nc';
{END_IF}

  _fbLoadProg           : Tc2_NCI.ItpLoadProgEx;

//Interpreter
  _fbReset              : Tc2_NCI.ItpResetEx2;
  _fbStartStop          : Tc2_NCI.ItpStartStopEx;
  _fbEStop              : Tc2_NCI.ItpEStopEx;
  _fbStepOnAfterEStop   : Tc2_NCI.ItpStepOnAfterEStopEx;

  _fbItpConfirmHsk      : Tc2_NCI.ItpConfirmHsk;
  _fbItpReadRParams     : Tc2_NCI.ItpReadRParamsEx;
  _fbItpWriteRParams    : Tc2_NCI.ItpWriteRParamsEx;
  _fbItpDelDtg          : Tc2_NCI.ItpDelDtgEx;

//ADS-Communication
  _fbReadLine           : Tc2_System.ADSREADEX;

// R Parameter
  // R[] Params used in G-Code
  // R[0..899]    local namespace of Channel
  // R[900..999]  global namespace of NC
  _pParameterRead       : POINTER TO ST_R_Parameter;
  _pParameterWrite      : POINTER TO ST_R_Parameter;
END_VAR

METHOD BuilDGroup : E_PROGRESS
VAR_INPUT
  Execute           : BOOL;
END_VAR
VAR_INST
  _eState           : E_PROGRESS;
  _rValue           : LREAL;
  _udiErr           : UDINT;
  _stMsg            : ST_Message;
END_VAR
IF NOT Check() THEN BuilDGroup := E_PROGRESS.PROGRESS_ERROR; RETURN; END_IF
IF NOT Execute THEN _eState := E_PROGRESS.PROGRESS_INIT; END_IF

CASE _eState
OF
  E_PROGRESS.PROGRESS_INIT:
    IF Execute 
    THEN
      _fbBuildGroup( 
                bExecute            := FALSE, 
                nGroupId            := ItpGetGroupId(sNciToPlc:=_NciChannelRef^.NcToPlc) , 
                nXAxisId            := _stCfgAxes^.nXAxisId,
                nYAxisId            := _stCfgAxes^.nYAxisId, 
                nZAxisId            := _stCfgAxes^.nZAxisId, 
                nQ1AxisId           := _stCfgAxes^.nQ1AxisId,
                nQ2AxisId           := _stCfgAxes^.nQ2AxisId, 
                nQ3AxisId           := _stCfgAxes^.nQ3AxisId, 
                nQ4AxisId           := _stCfgAxes^.nQ4AxisId, 
                nQ5AxisId           := _stCfgAxes^.nQ5AxisId);

      memset(ADR(_stMsg),0,SIZEOF(_stMsg));
      _udiErr                       := 0;
      _rValue                       := 0;
      _eState                       := E_PROGRESS.PROGRESS_BUSY;
    END_IF
END_CASE
CASE _eState
OF
  E_PROGRESS.PROGRESS_BUSY:
    _eState                         := E_PROGRESS.PROGRESS_STARTUP;
    _fbBuildGroup( 
                bExecute            := TRUE, 
                nGroupId            := ItpGetGroupId(sNciToPlc:=_NciChannelRef^.NcToPlc),
                  nErrId            => _udiErr);

    IF _fbBuildGroup.bErr 
    THEN
      _eState                       := E_PROGRESS.PROGRESS_ERROR;

      _stMsg.eType                  := E_MessageType.eMessageError;
      _stMsg.eDevice                := ChannelDevice;
      _stMsg.eSubdevice             := e_Subdevice.fbBuildGroup;
      _stMsg.iErrorNumber           := _fbBuildGroup.nErrId;
      _stMsg.sText                  := concat('BuildGroup Error: ', TO_STRING(_fbBuildGroup.nErrId));
      f_MessageSet(_stMsg);

    ELSE
      IF _fbBuildGroup.bBusy
      THEN
        _eState                     := E_PROGRESS.PROGRESS_STARTUP;

        _stMsg.eType                := E_MessageType.eMessageInfo;
        _stMsg.eDevice              := ChannelDevice;
        _stMsg.eSubdevice           := e_Subdevice.fbBuildGroup;
        _stMsg.iErrorNumber         := _fbBuildGroup.nGroupId;
        _stMsg.sText                := concat('BuildGroup Busy: ', TO_STRING(_fbBuildGroup.nGroupId));

        IF (_MessageLevel < E_MessageType.eMessageError)
        THEN
          f_MessageSet(_stMsg);
        END_IF
      END_IF
    END_IF
END_CASE
CASE _eState
OF
  E_PROGRESS.PROGRESS_STARTUP:
    _fbBuildGroup( 
                bExecute            := TRUE, 
                nGroupId            := ItpGetGroupId(sNciToPlc:=_NciChannelRef^.NcToPlc),
                  nErrId            => _udiErr);

    IF _fbBuildGroup.bErr 
    THEN
      _eState                       := E_PROGRESS.PROGRESS_ERROR;

      _stMsg.eType                  := E_MessageType.eMessageError;
      _stMsg.eDevice                := ChannelDevice;
      _stMsg.eSubdevice             := e_Subdevice.fbBuildGroup;
      _stMsg.iErrorNumber           := _fbBuildGroup.nErrId;
      _stMsg.sText                  := concat('BuildGroup Error: ', TO_STRING(_fbBuildGroup.nErrId));
      f_MessageSet(_stMsg);

    ELSE
      IF NOT _fbBuildGroup.bBusy
      THEN
        _eState                     := E_PROGRESS.PROGRESS_DONE;

        _stMsg.eType                := E_MessageType.eMessageInfo;
        _stMsg.eDevice              := ChannelDevice;
        _stMsg.eSubdevice           := e_Subdevice.fbBuildGroup;
        _stMsg.iErrorNumber         := _fbBuildGroup.nGroupId;
        _stMsg.sText                := concat('BuildGroup Done: ', TO_STRING(_fbBuildGroup.nGroupId));

        IF (_MessageLevel > E_MessageType.eMessageError)
        THEN
          f_MessageSet(_stMsg);
        END_IF
      END_IF
    END_IF
END_CASE
CASE _eState
OF
  E_PROGRESS.PROGRESS_ERROR,
  E_PROGRESS.PROGRESS_DONE:
    _fbBuildGroup( 
                bExecute            := FALSE, 
                nGroupId            := ItpGetGroupId(sNciToPlc:=_NciChannelRef^.NcToPlc));
END_CASE


BuilDGroup                          := _eState;
END_METHOD

(*
===============================================================
NCI-Group configured axes structure
===============================================================
*)
PROPERTY CfgAxes : POINTER TO ST_3D_Group
SET
_stCfgAxes := CfgAxes;  //Configured Group Axes
END_SET
END_PROPERTY

PROPERTY ChannelRef : POINTER TO ST_NciChannel_Ref
SET
_NciChannelRef := ChannelRef;
END_SET
END_PROPERTY

METHOD Check : BOOL
VAR
  _idx      : uint;
END_VAR
IF NOT NCI_ACTIVE
THEN
  _eCheck                         := E_CHECK_STATE.NCI_NOT_ACTIVATED;
  RETURN;
END_IF

IF NOT (_NciChannelRef <> 0)
THEN
  _eCheck                         := E_CHECK_STATE.NCI_CHANNEL_REF_POINTER_INVALID;
  RETURN;
END_IF

IF NOT (_NciChannelRef^.NcToPlc.ChnId <> 0)
THEN
  _eCheck                         := E_CHECK_STATE.NCI_CHANNEL_REF_POINTER_INVALID;
  RETURN;
END_IF

IF (_stCfgAxes <> 0)
THEN
  _eCheck                         := E_CHECK_STATE.NCI_AXIS_CONFIG_POINTER_INVALID;
  RETURN;
END_IF

IF NOT (_pParameterRead <> 0)
THEN
  _eCheck                         := E_CHECK_STATE.NCI_R_PARAMETER_READ_POINTER_INVALID;
  RETURN;
END_IF

IF NOT (_pParameterWrite <> 0)
THEN
  _eCheck                         := E_CHECK_STATE.NCI_R_PARAMETER_WRITE_POINTER_INVALID;
  RETURN;
END_IF

_eCheck                           := E_CHECK_STATE.CHECK_DONE;
Check                             := TRUE;
END_METHOD

METHOD ClearGroup : E_PROGRESS
VAR_INPUT
  Execute           : BOOL;
END_VAR
VAR_INST
  _eState           : E_PROGRESS;
  _rValue           : LREAL;
  _udiErr           : UDINT;
  _stMsg            : ST_Message;
END_VAR
IF NOT Check() THEN ClearGroup := E_PROGRESS.PROGRESS_ERROR; RETURN; END_IF
IF NOT Execute THEN _eState := E_PROGRESS.PROGRESS_INIT; END_IF

CASE _eState
OF
  E_PROGRESS.PROGRESS_INIT:
    IF Execute 
    THEN
      _fbClearGroup( 
                  bExecute          := FALSE, 
                  nGroupId          := ItpGetGroupId(sNciToPlc:= _NciChannelRef^.NcToPlc));

      memset(ADR(_stMsg),0,SIZEOF(_stMsg));
      _udiErr                       := 0;
      _rValue                       := 0;
      _eState                       := E_PROGRESS.PROGRESS_BUSY;
    END_IF
END_CASE
CASE _eState
OF
  E_PROGRESS.PROGRESS_BUSY:
    _eState                         := E_PROGRESS.PROGRESS_STARTUP;
    _fbClearGroup( 
                  bExecute          := TRUE, 
                  nGroupId          := ItpGetGroupId(sNciToPlc:= _NciChannelRef^.NcToPlc),
                  nErrId            => _udiErr);

    IF _fbClearGroup.bErr 
    THEN
      _eState                       := E_PROGRESS.PROGRESS_ERROR;

      _stMsg.eType                  := E_MessageType.eMessageError;
      _stMsg.eDevice                := ChannelDevice;
      _stMsg.eSubdevice             := e_Subdevice.fbClearGroup;
      _stMsg.iErrorNumber           := _fbClearGroup.nErrId;
      _stMsg.sText                  := concat('ClearGroup Error: ', TO_STRING(_fbClearGroup.nErrId));
      f_MessageSet(_stMsg);

    ELSE
      IF _fbClearGroup.bBusy
      THEN
        _eState                     := E_PROGRESS.PROGRESS_STARTUP;
        _stMsg.eType                := E_MessageType.eMessageInfo;
        _stMsg.eDevice              := ChannelDevice;
        _stMsg.eSubdevice           := e_Subdevice.fbClearGroup;
        _stMsg.iErrorNumber         := _fbClearGroup.nErrId;
        _stMsg.sText                := concat('ClearGroup Busy: ', TO_STRING(_fbClearGroup.nErrId));

        IF (_MessageLevel > E_MessageType.eMessageError)
        THEN
          f_MessageSet(_stMsg);
        END_IF
      END_IF
    END_IF
END_CASE
CASE _eState
OF
  E_PROGRESS.PROGRESS_STARTUP:
    _fbClearGroup( 
                  bExecute          := TRUE, 
                  nGroupId          := ItpGetGroupId(sNciToPlc:= _NciChannelRef^.NcToPlc),
                  nErrId            => _udiErr);

    IF _fbClearGroup.bErr 
    THEN
      _eState                       := E_PROGRESS.PROGRESS_ERROR;

      _stMsg.eType                  := E_MessageType.eMessageError;
      _stMsg.eDevice                := ChannelDevice;
      _stMsg.eSubdevice             := e_Subdevice.fbClearGroup;
      _stMsg.iErrorNumber           := _fbClearGroup.nErrId;
      _stMsg.sText                  := concat('ClearGroup Error: ', TO_STRING(_fbClearGroup.nErrId));
      f_MessageSet(_stMsg);

    ELSE
      IF NOT _fbClearGroup.bBusy
      THEN
        _eState                     := E_PROGRESS.PROGRESS_PREPARE;

        _stMsg.eType                := E_MessageType.eMessageInfo;
        _stMsg.eDevice              := ChannelDevice;
        _stMsg.eSubdevice           := e_Subdevice.fbClearGroup;
        _stMsg.iErrorNumber         := _fbClearGroup.nErrId;
        _stMsg.sText                := concat('ClearGroup Done: ', TO_STRING(_fbClearGroup.nErrId));

        IF (_MessageLevel > E_MessageType.eMessageError)
        THEN
          f_MessageSet(_stMsg);
        END_IF
      END_IF
    END_IF
END_CASE
CASE _eState
OF
  E_PROGRESS.PROGRESS_PREPARE:
    _eState                         := E_PROGRESS.PROGRESS_CHECK;
END_CASE
CASE _eState
OF
  E_PROGRESS.PROGRESS_CHECK:
    _eState                         := E_PROGRESS.PROGRESS_OCCUPIED;
END_CASE
CASE _eState
OF
  E_PROGRESS.PROGRESS_OCCUPIED:
    _eState                         := E_PROGRESS.PROGRESS_WORKING;
END_CASE
CASE _eState
OF
  E_PROGRESS.PROGRESS_WORKING:
    _eState                         := E_PROGRESS.PROGRESS_DONE;
END_CASE
CASE _eState
OF
  E_PROGRESS.PROGRESS_ERROR,
  E_PROGRESS.PROGRESS_DONE:
    _fbClearGroup( 
                  bExecute          := FALSE, 
                  nGroupId          := ItpGetGroupId(sNciToPlc:= _NciChannelRef^.NcToPlc));
END_CASE


ClearGroup                          := _eState;
END_METHOD

METHOD ConfirmHSK : E_PROGRESS
VAR_INPUT
  Execute           : BOOL;
END_VAR
VAR_INST
  _eState           : E_PROGRESS;
  _rValue           : LREAL;
  _udiErr           : UDINT;
  _stMsg            : ST_Message;
END_VAR
IF NOT Check() THEN ConfirmHSK := E_PROGRESS.PROGRESS_ERROR; RETURN; END_IF
IF NOT Execute THEN _eState := E_PROGRESS.PROGRESS_INIT; END_IF

CASE _eState
OF
  E_PROGRESS.PROGRESS_INIT:
    _NciChannelRef^.PlcToNc.MFuncGranted   := 0;

    IF Execute 
    THEN
      memset(ADR(_stMsg),0,SIZEOF(_stMsg));
      _udiErr                                 := 0;
      _rValue                                 := 0;
      _eState                                 := E_PROGRESS.PROGRESS_BUSY;
    END_IF
END_CASE
CASE _eState
OF
  E_PROGRESS.PROGRESS_BUSY:
    IF (_NciChannelRef^.PlcToNc.ChnAxesOvr > 0) AND NOT
       (_NciChannelRef^.NcToPlc.ChnState.8)
    THEN
      IF (_NciChannelRef^.NcToPlc.HskMFuncReq = 1)
      THEN
        _eState                               := E_PROGRESS.PROGRESS_STARTUP;

        _stMsg.eType                          := E_MessageType.eMessageInfo;
        _stMsg.eDevice                        := ChannelDevice;
        _stMsg.eSubdevice                     := e_Subdevice.fbConfirmHskItp;
        _stMsg.iErrorNumber                   := _NciChannelRef^.NcToPlc.HskMFuncNo;
        _stMsg.sText                          := concat('M Func check: ', 
                                                 TO_STRING(_NciChannelRef^.NcToPlc.HskMFuncNo));
        IF (_MessageLevel > E_MessageType.eMessageError)
        THEN
          f_MessageSet(_stMsg);
        END_IF
      END_IF
    END_IF
END_CASE
CASE _eState
OF
  E_PROGRESS.PROGRESS_STARTUP:
    _NciChannelRef^.PlcToNc.MFuncGranted   := 1;

    IF (_NciChannelRef^.NcToPlc.HskMFuncReq = 0)
    THEN
      _eState                                 := E_PROGRESS.PROGRESS_PREPARE;
      _NciChannelRef^.PlcToNc.MFuncGranted := 0;

      _stMsg.eType                            := E_MessageType.eMessageInfo;
      _stMsg.eDevice                          := ChannelDevice;
      _stMsg.eSubdevice                       := e_Subdevice.fbConfirmHskItp;
      _stMsg.iErrorNumber                     := _NciChannelRef^.NcToPlc.HskMFuncNo;
      _stMsg.sText                            := concat('M Func gone: ', 
                                               TO_STRING(_NciChannelRef^.NcToPlc.HskMFuncNo));
      IF (_MessageLevel > E_MessageType.eMessageError)
      THEN
        f_MessageSet(_stMsg);
      END_IF
    END_IF
END_CASE
CASE _eState
OF
  E_PROGRESS.PROGRESS_PREPARE:
    _eState                         := E_PROGRESS.PROGRESS_CHECK;
END_CASE
CASE _eState
OF
  E_PROGRESS.PROGRESS_CHECK:
    _eState                         := E_PROGRESS.PROGRESS_OCCUPIED;
END_CASE
CASE _eState
OF
  E_PROGRESS.PROGRESS_OCCUPIED:
    _eState                         := E_PROGRESS.PROGRESS_WORKING;
END_CASE
CASE _eState
OF
  E_PROGRESS.PROGRESS_WORKING:
    _eState                         := E_PROGRESS.PROGRESS_DONE;
END_CASE


ConfirmHSK                          := _eState;
END_METHOD

METHOD DeleteDistanceToGo : E_PROGRESS
VAR_INPUT
  Execute           : BOOL;
END_VAR
VAR_INST
  _eState           : E_PROGRESS;
  _rValue           : LREAL;
  _udiErr           : UDINT;
  _stMsg            : ST_Message;
END_VAR
IF NOT Check() THEN DeleteDistanceToGo := E_PROGRESS.PROGRESS_ERROR; RETURN; END_IF
IF NOT Execute THEN _eState := E_PROGRESS.PROGRESS_INIT; END_IF

CASE _eState
OF
  E_PROGRESS.PROGRESS_INIT:
    _fbItpDelDtg(
                sNciToPlc   := _NciChannelRef^.NcToPlc, 
                bExecute    := FALSE);

    IF Execute 
    THEN
      memset(ADR(_stMsg),0,SIZEOF(_stMsg));
      _udiErr                                 := 0;
      _rValue                                 := 0;
      _eState                                 := E_PROGRESS.PROGRESS_BUSY;
    END_IF
END_CASE
CASE _eState
OF
  E_PROGRESS.PROGRESS_BUSY:
    _fbItpDelDtg(
                sNciToPlc   := _NciChannelRef^.NcToPlc, 
                bExecute    := TRUE,
                nErrId      => _udiErr);

    IF _fbItpDelDtg.bErr 
    THEN
      _eState                       := E_PROGRESS.PROGRESS_ERROR;

      _stMsg.eType                  := E_MessageType.eMessageError;
      _stMsg.eDevice                := ChannelDevice;
      _stMsg.eSubdevice             := e_Subdevice.fbDelDtgItp;
      _stMsg.iErrorNumber           := _fbItpDelDtg.nErrId;
      _stMsg.sText                  := concat('Delete DistanceToGo Error: ', TO_STRING(_fbItpDelDtg.nErrId));
      f_MessageSet(_stMsg);

    ELSE
      IF _fbItpDelDtg.bBusy
      THEN
        _eState                     := E_PROGRESS.PROGRESS_STARTUP;

